C01818=1032.252,448.131,345.398,176.316,48.515,160.246
C01819=1032.229,447.887,345.444,176.296,48.510,160.242
C01820=1032.206,447.643,345.489,176.276,48.504,160.237
C01821=1032.183,447.398,345.535,176.258,48.499,160.233
C01822=1032.162,447.153,345.582,176.238,48.494,160.228
C01823=1032.140,446.909,345.629,176.219,48.489,160.224
C01824=1032.119,446.665,345.676,176.200,48.483,160.220
C01825=1032.099,446.420,345.724,176.181,48.478,160.215
C01826=1032.079,446.176,345.773,176.162,48.472,160.211
C01827=1032.060,445.932,345.821,176.143,48.467,160.206
C01828=1032.041,445.688,345.870,176.124,48.461,160.201
C01829=1032.022,445.444,345.920,176.106,48.455,160.197
C01830=1032.004,445.200,345.970,176.088,48.449,160.193
C01831=1031.987,444.957,346.020,176.069,48.443,160.188
C01832=1031.969,444.713,346.072,176.050,48.437,160.183
C01833=1031.953,444.468,346.122,176.033,48.431,160.179
C01834=1031.938,444.225,346.174,176.014,48.425,160.174
C01835=1031.921,443.982,346.226,175.996,48.419,160.170
C01836=1031.908,443.739,346.279,175.977,48.412,160.165
C01837=1031.892,443.495,346.332,175.960,48.406,160.161
C01838=1031.879,443.253,346.385,175.942,48.399,160.156
C01839=1031.864,443.010,346.438,175.924,48.393,160.152
C01840=1031.851,442.766,346.491,175.906,48.386,160.147
C01841=1031.838,442.521,346.545,175.889,48.379,160.142
C01842=1031.824,442.278,346.598,175.870,48.374,160.138
C01843=1031.810,442.034,346.652,175.853,48.367,160.133
C01844=1031.796,441.790,346.704,175.836,48.361,160.129
C01845=1031.783,441.546,346.758,175.818,48.354,160.125
C01846=1031.769,441.302,346.810,175.801,48.347,160.120
C01847=1031.755,441.058,346.864,175.784,48.341,160.116
C01848=1031.742,440.814,346.916,175.766,48.335,160.111
C01849=1031.728,440.570,346.970,175.749,48.329,160.107
C01850=1031.715,440.326,347.023,175.732,48.322,160.103
C01851=1031.702,440.082,347.075,175.715,48.316,160.098
C01852=1031.688,439.838,347.129,175.698,48.310,160.094
C01853=1031.675,439.594,347.180,175.681,48.304,160.090
C01854=1031.662,439.350,347.234,175.664,48.297,160.085
C01855=1031.648,439.106,347.286,175.646,48.291,160.081
C01856=1031.634,438.844,347.343,175.629,48.284,160.076
C01857=1031.620,438.582,347.399,175.611,48.278,160.072
C01858=1031.606,438.319,347.456,175.593,48.271,160.067
C01859=1031.591,438.057,347.511,175.575,48.265,160.063
C01860=1031.578,437.813,347.564,175.559,48.258,160.059
C01861=1031.565,437.569,347.615,175.542,48.253,160.054
C01862=1031.552,437.324,347.668,175.526,48.246,160.050
C01863=1031.539,437.080,347.720,175.509,48.241,160.046
C01864=1031.526,436.836,347.772,175.494,48.234,160.042
C01865=1031.513,436.592,347.824,175.477,48.229,160.038
C01866=1031.500,436.347,347.876,175.461,48.222,160.034
C01867=1031.487,436.103,347.928,175.444,48.217,160.030
C01868=1031.474,435.859,347.979,175.429,48.211,160.026
C01869=1031.462,435.615,348.031,175.413,48.205,160.022
C01870=1031.448,435.370,348.083,175.396,48.199,160.018
C01871=1031.436,435.126,348.134,175.381,48.193,160.014
C01872=1031.423,434.882,348.186,175.365,48.187,160.010
C01873=1031.410,434.637,348.237,175.350,48.182,160.006
C01874=1031.398,434.392,348.289,175.334,48.176,160.002
C01875=1031.385,434.149,348.340,175.317,48.170,159.998
C01876=1031.366,433.797,348.414,175.296,48.162,159.992
C01877=1031.348,433.447,348.487,175.273,48.154,159.987
C01878=1031.330,433.095,348.560,175.251,48.145,159.981
C01879=1031.312,432.744,348.634,175.229,48.137,159.976
C01880=1031.299,432.500,348.685,175.214,48.132,159.972
C01881=1031.287,432.256,348.735,175.198,48.126,159.968
C01882=1031.274,432.011,348.786,175.183,48.121,159.965
C01883=1031.262,431.766,348.837,175.168,48.115,159.961
C01884=1031.249,431.521,348.888,175.153,48.110,159.957
C01885=1031.237,431.277,348.938,175.137,48.104,159.953
C01886=1031.224,431.032,348.989,175.123,48.098,159.950
C01887=1031.212,430.788,349.039,175.108,48.093,159.946
C01888=1031.199,430.543,349.090,175.093,48.087,159.942
C01889=1031.187,430.299,349.140,175.078,48.082,159.938
C01890=1031.175,430.054,349.191,175.064,48.077,159.935
C01891=1031.163,429.809,349.242,175.049,48.071,159.931
C01892=1031.151,429.565,349.291,175.033,48.066,159.928
C01893=1031.139,429.320,349.341,175.019,48.061,159.924
C01894=1031.126,429.076,349.392,175.004,48.055,159.920
C01895=1031.114,428.831,349.442,174.990,48.050,159.917
C01896=1031.102,428.586,349.493,174.976,48.045,159.913
C01897=1031.091,428.342,349.543,174.961,48.039,159.910
C01898=1031.078,428.097,349.593,174.946,48.034,159.906
C01899=1031.066,427.852,349.643,174.933,48.029,159.903
C01900=1031.055,427.608,349.692,174.919,48.023,159.899
C01901=1031.042,427.363,349.742,174.904,48.019,159.896
C01902=1031.030,427.118,349.792,174.890,48.013,159.892
C01903=1031.019,426.874,349.842,174.876,48.008,159.889
C01904=1031.007,426.628,349.892,174.861,48.003,159.885
C01905=1030.995,426.383,349.942,174.847,47.998,159.882
C01906=1030.983,426.139,349.991,174.834,47.993,159.878
C01907=1030.971,425.893,350.040,174.819,47.988,159.875
C01908=1030.959,425.649,350.089,174.805,47.983,159.872
C01909=1030.947,425.404,350.139,174.791,47.978,159.868
C01910=1030.935,425.159,350.188,174.778,47.972,159.865
C01911=1030.923,424.914,350.238,174.764,47.967,159.861
C01912=1030.913,424.705,350.280,174.752,47.963,159.859
C01913=1030.903,424.497,350.322,174.740,47.959,159.856
C01914=1030.893,424.288,350.364,174.729,47.955,159.853
C01915=1030.883,424.079,350.406,174.717,47.950,159.850
C01916=1030.874,423.871,350.447,174.706,47.947,159.847
C01917=1030.864,423.662,350.489,174.693,47.942,159.845
C01918=1030.854,423.453,350.531,174.682,47.938,159.842
C01919=1030.844,423.244,350.572,174.671,47.934,159.839
C01920=1030.833,422.999,350.621,174.657,47.929,159.836
C01921=1030.821,422.753,350.670,174.644,47.924,159.833
C01922=1030.809,422.509,350.720,174.630,47.920,159.829
C01923=1030.797,422.264,350.767,174.617,47.914,159.826
C01924=1030.786,422.019,350.816,174.604,47.910,159.823
C01925=1030.775,421.773,350.865,174.591,47.905,159.820
C01926=1030.763,421.529,350.913,174.578,47.900,159.817
C01927=1030.751,421.283,350.962,174.564,47.896,159.813
C01928=1030.740,421.038,351.011,174.551,47.891,159.810
C01929=1030.729,420.793,351.059,174.539,47.886,159.807
C01930=1030.717,420.548,351.107,174.525,47.882,159.804
C01931=1030.705,420.303,351.156,174.512,47.877,159.801
C01932=1030.695,420.058,351.204,174.499,47.872,159.798
C01933=1030.683,419.813,351.251,174.486,47.867,159.795
C01934=1030.672,419.568,351.300,174.473,47.863,159.792
C01935=1030.661,419.323,351.348,174.461,47.858,159.789
C01936=1030.649,419.078,351.396,174.447,47.854,159.786
C01937=1030.638,418.832,351.444,174.434,47.850,159.783
C01938=1030.627,418.587,351.492,174.422,47.845,159.779
C01939=1030.616,418.342,351.539,174.409,47.841,159.777
C01940=1030.604,418.097,351.588,174.397,47.836,159.773
C01941=1030.593,417.852,351.636,174.384,47.831,159.771
C01942=1030.582,417.607,351.683,174.372,47.827,159.768
C01943=1030.571,417.361,351.731,174.359,47.822,159.765
C01944=1030.560,417.116,351.779,174.346,47.818,159.762
C01945=1030.549,416.872,351.827,174.334,47.814,159.759
C01946=1030.538,416.626,351.874,174.322,47.809,159.756
C01947=1030.527,416.380,351.923,174.310,47.805,159.753
C01948=1030.516,416.135,351.969,174.298,47.801,159.750
C01949=1030.505,415.890,352.017,174.285,47.796,159.747
C01950=1030.494,415.645,352.064,174.273,47.792,159.744
C01951=1030.483,415.399,352.111,174.261,47.788,159.741
C01952=1030.472,415.154,352.158,174.248,47.783,159.739
C01953=1030.461,414.909,352.206,174.236,47.780,159.736
C01954=1030.450,414.664,352.253,174.224,47.775,159.733
C01955=1030.439,414.418,352.300,174.212,47.771,159.730
C01956=1030.428,414.173,352.347,174.199,47.767,159.727
C01957=1030.418,413.928,352.394,174.187,47.763,159.725
C01958=1030.406,413.682,352.441,174.175,47.758,159.722
C01959=1030.396,413.437,352.488,174.164,47.754,159.719
C01960=1030.385,413.192,352.535,174.152,47.750,159.716
C01961=1030.374,412.947,352.581,174.140,47.746,159.713
C01962=1030.363,412.701,352.629,174.128,47.742,159.711
C01963=1030.352,412.456,352.676,174.116,47.737,159.708
C01964=1030.343,412.210,352.722,174.105,47.733,159.705
C01965=1030.332,411.965,352.769,174.093,47.730,159.703
C01966=1030.321,411.720,352.815,174.082,47.726,159.700
C01967=1030.310,411.473,352.862,174.070,47.722,159.697
C01968=1030.299,411.229,352.909,174.058,47.717,159.694
C01969=1030.289,410.983,352.956,174.046,47.713,159.692
C01970=1030.278,410.738,353.002,174.035,47.709,159.689
C01971=1030.268,410.492,353.049,174.023,47.705,159.686
C01972=1030.258,410.247,353.095,174.012,47.702,159.684
C01973=1030.247,410.001,353.141,174.000,47.698,159.681
C01974=1030.236,409.756,353.187,173.989,47.694,159.679
C01975=1030.226,409.510,353.233,173.977,47.690,159.676
C01976=1030.215,409.241,353.284,173.965,47.686,159.673
C01977=1030.203,408.972,353.334,173.952,47.682,159.670
C01978=1030.191,408.703,353.385,173.940,47.677,159.668
C01979=1030.180,408.433,353.435,173.928,47.674,159.665
C01980=1030.169,408.188,353.481,173.916,47.670,159.662
C01981=1030.158,407.942,353.527,173.906,47.666,159.660
C01982=1030.148,407.696,353.572,173.894,47.662,159.657
C01983=1030.137,407.451,353.618,173.883,47.659,159.655
C01984=1030.127,407.205,353.664,173.871,47.655,159.652
C01985=1030.117,406.960,353.710,173.861,47.651,159.650
C01986=1030.106,406.715,353.756,173.850,47.648,159.647
C01987=1030.096,406.468,353.802,173.838,47.644,159.645
C01988=1030.086,406.223,353.847,173.828,47.640,159.642
C01989=1030.076,405.978,353.893,173.817,47.637,159.640
C01990=1030.065,405.732,353.938,173.806,47.633,159.637
C01991=1030.055,405.487,353.984,173.795,47.629,159.635
C01992=1030.045,405.240,354.029,173.784,47.626,159.633
C01993=1030.035,404.996,354.074,173.773,47.622,159.630
C01994=1030.025,404.749,354.120,173.762,47.619,159.628
C01995=1030.015,404.504,354.165,173.752,47.615,159.625
C01996=1030.004,404.258,354.210,173.741,47.612,159.623
C01997=1029.994,404.013,354.256,173.730,47.608,159.620
C01998=1029.984,403.767,354.301,173.719,47.605,159.618
C01999=1029.974,403.522,354.346,173.709,47.601,159.616
C02000=1029.964,403.276,354.392,173.699,47.598,159.613
C02001=1029.954,403.031,354.437,173.688,47.594,159.611
C02002=1029.944,402.785,354.481,173.677,47.590,159.609
C02003=1029.934,402.539,354.527,173.666,47.588,159.606
C02004=1029.924,402.293,354.571,173.656,47.584,159.604
C02005=1029.915,402.048,354.616,173.646,47.581,159.602
C02006=1029.904,401.802,354.661,173.635,47.577,159.599
C02007=1029.894,401.556,354.706,173.625,47.574,159.597
C02008=1029.885,401.311,354.751,173.615,47.570,159.595
C02009=1029.874,401.064,354.796,173.604,47.567,159.593
C02010=1029.865,400.819,354.841,173.594,47.564,159.590
C02011=1029.855,400.573,354.886,173.583,47.560,159.588
C02012=1029.846,400.327,354.930,173.573,47.557,159.586
C02013=1029.835,400.082,354.974,173.563,47.554,159.584
C02014=1029.825,399.836,355.019,173.552,47.550,159.581
C02015=1029.815,399.590,355.064,173.542,47.547,159.579
C02016=1029.806,399.344,355.108,173.531,47.544,159.577
C02017=1029.795,399.099,355.153,173.521,47.541,159.575
C02018=1029.786,398.853,355.197,173.512,47.538,159.572
C02019=1029.776,398.607,355.242,173.502,47.535,159.570
C02020=1029.767,398.361,355.286,173.492,47.532,159.568
C02021=1029.757,398.115,355.329,173.482,47.528,159.566
C02022=1029.747,397.870,355.374,173.471,47.525,159.564
C02023=1029.737,397.624,355.418,173.461,47.523,159.562
C02024=1029.727,397.378,355.462,173.451,47.520,159.560
C02025=1029.718,397.132,355.506,173.441,47.516,159.557
C02026=1029.707,396.886,355.550,173.431,47.513,159.555
C02027=1029.698,396.640,355.594,173.422,47.510,159.553
C02028=1029.689,396.394,355.638,173.412,47.507,159.551
C02029=1029.678,396.148,355.682,173.402,47.504,159.549
C02030=1029.670,395.903,355.725,173.392,47.501,159.547
C02031=1029.660,395.657,355.770,173.382,47.498,159.545
C02032=1029.650,395.411,355.813,173.373,47.495,159.543
C02033=1029.641,395.165,355.857,173.363,47.492,159.541
C02034=1029.631,394.919,355.901,173.353,47.490,159.539
C02035=1029.622,394.674,355.944,173.343,47.486,159.536
C02036=1029.611,394.425,355.989,173.334,47.484,159.534
C02037=1029.602,394.178,356.033,173.324,47.480,159.532
C02038=1029.593,393.930,356.077,173.314,47.478,159.530
C02039=1029.583,393.683,356.120,173.304,47.475,159.528
C02040=1029.574,393.436,356.164,173.295,47.472,159.526
C02041=1029.564,393.190,356.207,173.285,47.469,159.524
C02042=1029.555,392.944,356.250,173.276,47.467,159.522
C02043=1029.545,392.698,356.294,173.266,47.464,159.520
C02044=1029.535,392.452,356.337,173.256,47.461,159.518
C02045=1029.527,392.206,356.380,173.247,47.459,159.516
C02046=1029.517,391.960,356.423,173.238,47.455,159.514
C02047=1029.508,391.714,356.467,173.228,47.452,159.512
C02048=1029.498,391.468,356.510,173.219,47.450,159.510
C02049=1029.489,391.223,356.554,173.209,47.447,159.508
C02050=1029.479,390.976,356.596,173.200,47.445,159.506
C02051=1029.470,390.730,356.639,173.191,47.442,159.505
C02052=1029.461,390.484,356.683,173.182,47.439,159.503
C02053=1029.452,390.239,356.725,173.172,47.436,159.501
C02054=1029.442,389.992,356.769,173.162,47.434,159.499
C02055=1029.433,389.746,356.811,173.154,47.431,159.497
C02056=1029.423,389.500,356.854,173.145,47.429,159.495
C02057=1029.415,389.254,356.897,173.135,47.426,159.493
C02058=1029.405,389.007,356.940,173.126,47.423,159.491
C02059=1029.396,388.761,356.982,173.117,47.421,159.489
C02060=1029.387,388.516,357.025,173.108,47.418,159.487
C02061=1029.377,388.269,357.068,173.098,47.416,159.486
C02062=1029.368,388.023,357.110,173.090,47.413,159.484
C02063=1029.359,387.777,357.153,173.080,47.411,159.482
C02064=1029.350,387.531,357.196,173.072,47.408,159.480
C02065=1029.341,387.285,357.239,173.063,47.406,159.478
C02066=1029.332,387.038,357.280,173.053,47.403,159.476
C02067=1029.322,386.793,357.323,173.045,47.401,159.475
C02068=1029.313,386.546,357.366,173.036,47.399,159.473
C02069=1029.304,386.300,357.408,173.027,47.396,159.471
C02070=1029.295,386.054,357.450,173.018,47.393,159.469
C02071=1029.286,385.807,357.492,173.008,47.391,159.467
C02072=1029.276,385.561,357.535,173.000,47.389,159.466
C02073=1029.267,385.315,357.577,172.991,47.387,159.464
C02074=1029.258,385.069,357.619,172.983,47.384,159.462
C02075=1029.249,384.823,357.661,172.973,47.382,159.460
C02076=1029.240,384.576,357.702,172.965,47.380,159.459
C02077=1029.231,384.330,357.745,172.956,47.377,159.457
C02078=1029.222,384.084,357.787,172.948,47.375,159.455
C02079=1029.213,383.838,357.828,172.938,47.373,159.453
C02080=1029.203,383.591,357.871,172.930,47.371,159.452
C02081=1029.194,383.345,357.913,172.921,47.368,159.450
C02082=1029.186,383.099,357.955,172.913,47.366,159.448
C02083=1029.177,382.852,357.996,172.903,47.364,159.446
C02084=1029.168,382.606,358.038,172.895,47.361,159.445
C02085=1029.159,382.359,358.080,172.887,47.359,159.443
C02086=1029.150,382.113,358.121,172.878,47.357,159.442
C02087=1029.141,381.867,358.163,172.870,47.355,159.440
C02088=1029.133,381.621,358.205,172.860,47.353,159.438
C02089=1029.124,381.375,358.246,172.852,47.350,159.436
C02090=1029.115,381.128,358.288,172.844,47.348,159.435
C02091=1029.106,380.882,358.330,172.835,47.346,159.433
C02092=1029.097,380.653,358.369,172.827,47.344,159.432
C02093=1029.089,380.424,358.407,172.819,47.343,159.430
C02094=1029.081,380.196,358.446,172.812,47.340,159.429
C02095=1029.072,379.967,358.484,172.804,47.339,159.427
C02096=1029.065,379.737,358.522,172.796,47.337,159.426
C02097=1029.056,379.509,358.561,172.788,47.335,159.424
C02098=1029.048,379.279,358.599,172.780,47.332,159.422
C02099=1029.040,379.050,358.638,172.772,47.331,159.421
C02100=1029.031,378.804,358.679,172.764,47.329,159.419
C02101=1029.022,378.557,358.721,172.756,47.327,159.418
C02102=1029.014,378.311,358.762,172.748,47.324,159.416
C02103=1029.005,378.065,358.803,172.739,47.323,159.415
C02104=1028.996,377.818,358.845,172.731,47.321,159.413
C02105=1028.988,377.572,358.886,172.723,47.318,159.411
C02106=1028.979,377.326,358.927,172.715,47.317,159.410
C02107=1028.971,377.079,358.968,172.707,47.315,159.408
C02108=1028.962,376.832,359.009,172.698,47.313,159.407
C02109=1028.953,376.586,359.050,172.690,47.311,159.405
C02110=1028.944,376.339,359.091,172.682,47.309,159.404
C02111=1028.936,376.094,359.131,172.674,47.307,159.402
C02112=1028.927,375.847,359.172,172.666,47.306,159.401
C02113=1028.918,375.600,359.213,172.658,47.304,159.399
C02114=1028.909,375.354,359.254,172.650,47.302,159.398
C02115=1028.901,375.107,359.295,172.642,47.300,159.396
C02116=1028.893,374.861,359.336,172.634,47.298,159.395
C02117=1028.883,374.614,359.376,172.626,47.296,159.393
C02118=1028.875,374.368,359.417,172.618,47.294,159.392
C02119=1028.867,374.121,359.458,172.610,47.293,159.390
C02120=1028.858,373.875,359.498,172.602,47.291,159.389
C02121=1028.849,373.628,359.539,172.594,47.289,159.387
C02122=1028.840,373.382,359.579,172.586,47.288,159.386
C02123=1028.832,373.135,359.620,172.578,47.286,159.384
C02124=1028.824,372.889,359.660,172.570,47.284,159.383
C02125=1028.815,372.641,359.700,172.562,47.282,159.381
C02126=1028.807,372.395,359.741,172.554,47.281,159.380
C02127=1028.799,372.149,359.781,172.546,47.279,159.378
C02128=1028.789,371.902,359.822,172.538,47.277,159.377
C02129=1028.781,371.656,359.862,172.531,47.276,159.376
C02130=1028.774,371.409,359.902,172.523,47.274,159.374
C02131=1028.764,371.162,359.943,172.515,47.273,159.373
C02132=1028.756,370.916,359.983,172.507,47.271,159.371
C02133=1028.748,370.669,360.023,172.500,47.269,159.370
C02134=1028.740,370.423,360.063,172.492,47.267,159.368
C02135=1028.731,370.176,360.104,172.484,47.266,159.367
C02136=1028.723,369.930,360.144,172.476,47.264,159.366
C02137=1028.715,369.683,360.184,172.469,47.263,159.364
C02138=1028.706,369.437,360.224,172.462,47.261,159.363
C02139=1028.698,369.190,360.264,172.454,47.259,159.361
C02140=1028.690,368.943,360.304,172.447,47.258,159.360
C02141=1028.681,368.696,360.344,172.439,47.256,159.359
C02142=1028.673,368.450,360.384,172.431,47.255,159.357
C02143=1028.665,368.203,360.424,172.423,47.253,159.356
C02144=1028.656,367.956,360.463,172.416,47.252,159.355
C02145=1028.647,367.709,360.503,172.408,47.251,159.353
C02146=1028.639,367.463,360.542,172.400,47.249,159.352
C02147=1028.631,367.217,360.583,172.393,47.248,159.351
C02148=1028.622,366.970,360.622,172.385,47.246,159.349
C02149=1028.614,366.723,360.661,172.378,47.245,159.348
C02150=1028.606,366.477,360.701,172.371,47.243,159.347
C02151=1028.598,366.230,360.741,172.363,47.242,159.345
C02152=1028.590,366.011,360.775,172.357,47.241,159.344
C02153=1028.583,365.792,360.811,172.350,47.239,159.343
C02154=1028.575,365.574,360.845,172.343,47.239,159.342
C02155=1028.568,365.356,360.880,172.337,47.238,159.341
C02156=1028.561,365.137,360.916,172.330,47.236,159.340
C02157=1028.553,364.919,360.951,172.324,47.235,159.339
C02158=1028.546,364.701,360.985,172.317,47.233,159.337
C02159=1028.539,364.482,361.020,172.311,47.232,159.336
C02160=1028.531,364.235,361.060,172.303,47.231,159.335
C02161=1028.522,363.988,361.099,172.296,47.230,159.334
C02162=1028.515,363.742,361.139,172.289,47.229,159.333
C02163=1028.506,363.494,361.177,172.282,47.227,159.331
C02164=1028.498,363.248,361.217,172.274,47.226,159.330
C02165=1028.490,363.002,361.256,172.267,47.225,159.329
C02166=1028.483,362.754,361.295,172.260,47.224,159.328
C02167=1028.474,362.508,361.334,172.253,47.222,159.326
C02168=1028.466,362.261,361.373,172.245,47.221,159.325
C02169=1028.458,362.014,361.413,172.238,47.220,159.324
C02170=1028.450,361.767,361.452,172.231,47.219,159.323
C02171=1028.442,361.521,361.491,172.224,47.217,159.321
C02172=1028.434,361.274,361.530,172.217,47.217,159.320
C02173=1028.426,361.027,361.570,172.210,47.215,159.319
C02174=1028.418,360.780,361.608,172.203,47.214,159.318
C02175=1028.410,360.533,361.647,172.195,47.213,159.316
C02176=1028.402,360.287,361.686,172.189,47.212,159.315
C02177=1028.394,360.039,361.724,172.181,47.211,159.314
C02178=1028.385,359.793,361.764,172.174,47.210,159.313
C02179=1028.377,359.546,361.802,172.167,47.208,159.312
C02180=1028.370,359.299,361.840,172.160,47.207,159.311
C02181=1028.362,359.052,361.879,172.153,47.207,159.309
C02182=1028.353,358.805,361.918,172.146,47.205,159.308
C02183=1028.346,358.559,361.957,172.139,47.204,159.307
C02184=1028.337,358.312,361.995,172.132,47.204,159.306
C02185=1028.329,358.064,362.034,172.125,47.202,159.305
C02186=1028.322,357.818,362.072,172.118,47.201,159.304
C02187=1028.314,357.571,362.111,172.111,47.200,159.303
C02188=1028.305,357.323,362.149,172.104,47.199,159.301
C02189=1028.298,357.077,362.188,172.097,47.199,159.300
C02190=1028.290,356.830,362.226,172.091,47.198,159.299
C02191=1028.282,356.583,362.264,172.083,47.196,159.298
C02192=1028.273,356.336,362.302,172.077,47.195,159.297
C02193=1028.265,356.089,362.341,172.069,47.195,159.296
C02194=1028.258,355.843,362.379,172.063,47.193,159.295
C02195=1028.249,355.595,362.418,172.056,47.193,159.294
C02196=1028.242,355.349,362.456,172.050,47.192,159.293
C02197=1028.234,355.102,362.495,172.042,47.191,159.291
C02198=1028.226,354.854,362.532,172.036,47.190,159.290
C02199=1028.218,354.607,362.571,172.029,47.189,159.289
C02200=1028.210,354.361,362.609,172.021,47.188,159.288
C02201=1028.202,354.114,362.647,172.015,47.187,159.287
C02202=1028.195,353.867,362.685,172.008,47.187,159.286
C02203=1028.186,353.619,362.723,172.002,47.186,159.285
C02204=1028.178,353.373,362.760,171.995,47.185,159.284
C02205=1028.171,353.126,362.798,171.988,47.184,159.283
C02206=1028.163,352.879,362.837,171.981,47.184,159.282
C02207=1028.156,352.632,362.875,171.975,47.183,159.281
C02208=1028.147,352.385,362.913,171.968,47.182,159.280
C02209=1028.139,352.138,362.950,171.962,47.181,159.279
C02210=1028.132,351.891,362.988,171.955,47.180,159.278
C02211=1028.124,351.643,363.026,171.948,47.180,159.277
C02212=1028.117,351.429,363.059,171.942,47.179,159.276
C02213=1028.111,351.213,363.092,171.937,47.178,159.275
C02214=1028.103,350.998,363.125,171.931,47.178,159.274
C02215=1028.097,350.782,363.158,171.925,47.178,159.273
C02216=1028.090,350.568,363.190,171.919,47.177,159.272
C02217=1028.083,350.352,363.223,171.914,47.176,159.271
C02218=1028.076,350.137,363.256,171.908,47.175,159.270
C02219=1028.070,349.922,363.289,171.902,47.175,159.269
C02220=1028.063,349.675,363.327,171.896,47.174,159.269
C02221=1028.054,349.428,363.364,171.890,47.173,159.268
C02222=1028.047,349.180,363.402,171.882,47.173,159.266
C02223=1028.040,348.933,363.439,171.877,47.172,159.266
C02224=1028.032,348.686,363.476,171.870,47.172,159.265
C02225=1028.024,348.440,363.515,171.863,47.171,159.264
C02226=1028.015,348.192,363.552,171.857,47.171,159.263
C02227=1028.008,347.945,363.589,171.850,47.170,159.262
C02228=1028.000,347.698,363.626,171.844,47.169,159.261
C02229=1027.993,347.451,363.664,171.838,47.169,159.260
C02230=1027.985,347.204,363.701,171.831,47.168,159.259
C02231=1027.977,346.957,363.739,171.825,47.168,159.258
C02232=1027.969,346.710,363.776,171.819,47.167,159.257
C02233=1027.962,346.463,363.813,171.812,47.166,159.256
C02234=1027.954,346.215,363.849,171.806,47.166,159.255
C02235=1027.947,345.968,363.887,171.800,47.166,159.254
C02236=1027.939,345.721,363.924,171.793,47.165,159.253
C02237=1027.932,345.474,363.961,171.787,47.165,159.252
C02238=1027.924,345.227,363.998,171.780,47.164,159.251
C02239=1027.917,344.980,364.036,171.774,47.164,159.250
C02240=1027.909,344.733,364.072,171.768,47.163,159.249
C02241=1027.901,344.486,364.109,171.762,47.163,159.249
C02242=1027.894,344.239,364.146,171.755,47.163,159.248
C02243=1027.886,343.991,364.183,171.749,47.162,159.247
C02244=1027.879,343.744,364.220,171.743,47.162,159.246
C02245=1027.871,343.497,364.257,171.737,47.161,159.245
C02246=1027.864,343.250,364.294,171.730,47.161,159.244
C02247=1027.856,343.003,364.331,171.724,47.161,159.243
C02248=1027.848,342.755,364.367,171.718,47.160,159.242
C02249=1027.841,342.508,364.405,171.712,47.160,159.241
C02250=1027.833,342.261,364.442,171.705,47.160,159.241
C02251=1027.825,342.014,364.478,171.699,47.159,159.240
C02252=1027.818,341.766,364.515,171.693,47.159,159.239
C02253=1027.810,341.519,364.552,171.687,47.158,159.238
C02254=1027.803,341.272,364.588,171.681,47.158,159.237
C02255=1027.795,341.025,364.625,171.674,47.158,159.236
C02256=1027.788,340.777,364.661,171.668,47.157,159.235
C02257=1027.780,340.531,364.698,171.662,47.157,159.234
C02258=1027.773,340.283,364.735,171.656,47.157,159.234
C02259=1027.766,340.036,364.771,171.651,47.156,159.233
C02260=1027.758,339.789,364.807,171.644,47.156,159.232
C02261=1027.750,339.542,364.844,171.638,47.156,159.231
C02262=1027.742,339.294,364.880,171.632,47.156,159.230
C02263=1027.735,339.048,364.916,171.626,47.155,159.229
C02264=1027.728,338.800,364.953,171.620,47.155,159.229
C02265=1027.721,338.552,364.989,171.613,47.155,159.228
C02266=1027.713,338.305,365.026,171.607,47.155,159.227
C02267=1027.705,338.057,365.062,171.602,47.155,159.226
C02268=1027.698,337.811,365.098,171.596,47.155,159.225
C02269=1027.690,337.564,365.135,171.590,47.154,159.225
C02270=1027.683,337.316,365.171,171.584,47.154,159.224
C02271=1027.675,337.069,365.207,171.577,47.154,159.223
C02272=1027.669,336.852,365.238,171.573,47.154,159.222
C02273=1027.662,336.636,365.270,171.567,47.154,159.222
C02274=1027.656,336.418,365.302,171.562,47.154,159.221
C02275=1027.649,336.202,365.333,171.556,47.154,159.220
C02276=1027.643,335.985,365.366,171.552,47.153,159.219
C02277=1027.637,335.768,365.396,171.546,47.154,159.219
C02278=1027.630,335.552,365.429,171.541,47.154,159.218
C02279=1027.624,335.334,365.460,171.536,47.154,159.217
C02280=1027.616,335.087,365.496,171.530,47.153,159.217
C02281=1027.610,334.840,365.532,171.524,47.153,159.216
C02282=1027.602,334.592,365.568,171.518,47.154,159.215
C02283=1027.595,334.346,365.604,171.512,47.153,159.214
C02284=1027.587,334.098,365.640,171.507,47.153,159.214
C02285=1027.580,333.850,365.676,171.501,47.153,159.213
C02286=1027.573,333.603,365.712,171.495,47.153,159.212
C02287=1027.565,333.355,365.747,171.490,47.153,159.211
C02288=1027.558,333.109,365.783,171.484,47.153,159.211
C02289=1027.550,332.861,365.819,171.478,47.153,159.210
C02290=1027.543,332.614,365.854,171.472,47.153,159.209
C02291=1027.535,332.367,365.890,171.466,47.153,159.208
C02292=1027.529,332.119,365.925,171.460,47.153,159.208
C02293=1027.521,331.872,365.962,171.454,47.154,159.207
C02294=1027.514,331.624,365.997,171.449,47.154,159.206
C02295=1027.506,331.377,366.032,171.443,47.153,159.205
C02296=1027.499,331.130,366.067,171.437,47.153,159.205
C02297=1027.491,330.883,366.104,171.431,47.154,159.204
C02298=1027.485,330.635,366.139,171.426,47.154,159.203
C02299=1027.477,330.388,366.175,171.420,47.154,159.203
C02300=1027.470,330.140,366.210,171.414,47.154,159.202
C02301=1027.462,329.893,366.245,171.409,47.154,159.201
C02302=1027.455,329.646,366.281,171.403,47.154,159.201
C02303=1027.448,329.398,366.316,171.397,47.154,159.200
C02304=1027.441,329.150,366.352,171.392,47.155,159.199
C02305=1027.434,328.904,366.387,171.386,47.155,159.199
C02306=1027.426,328.656,366.422,171.380,47.155,159.198
C02307=1027.419,328.409,366.457,171.375,47.155,159.197
C02308=1027.412,328.161,366.493,171.369,47.155,159.197
C02309=1027.404,327.914,366.529,171.363,47.155,159.196
C02310=1027.398,327.666,366.564,171.358,47.155,159.195
C02311=1027.390,327.419,366.598,171.352,47.156,159.194
C02312=1027.383,327.171,366.634,171.347,47.156,159.194
C02313=1027.375,326.924,366.668,171.341,47.157,159.193
C02314=1027.368,326.677,366.704,171.336,47.157,159.193
C02315=1027.360,326.429,366.739,171.330,47.157,159.192
C02316=1027.353,326.182,366.773,171.325,47.158,159.191
C02317=1027.346,325.935,366.808,171.319,47.158,159.191
C02318=1027.338,325.687,366.843,171.313,47.158,159.190
C02319=1027.331,325.440,366.878,171.308,47.159,159.190
C02320=1027.324,325.192,366.912,171.302,47.159,159.189
C02321=1027.316,324.944,366.947,171.297,47.159,159.188
C02322=1027.309,324.697,366.982,171.291,47.160,159.188
C02323=1027.302,324.450,367.017,171.286,47.160,159.187
C02324=1027.295,324.202,367.052,171.280,47.161,159.186
C02325=1027.287,323.954,367.086,171.275,47.161,159.186
C02326=1027.280,323.707,367.120,171.269,47.161,159.185
C02327=1027.273,323.460,367.156,171.264,47.162,159.185
C02328=1027.265,323.213,367.190,171.258,47.162,159.184
C02329=1027.259,322.965,367.225,171.253,47.163,159.183
C02330=1027.251,322.717,367.259,171.247,47.163,159.183
C02331=1027.243,322.470,367.294,171.243,47.163,159.182
C02332=1027.237,322.250,367.325,171.237,47.163,159.182
C02333=1027.231,322.031,367.356,171.233,47.164,159.181
C02334=1027.224,321.812,367.386,171.227,47.165,159.181
C02335=1027.218,321.593,367.416,171.223,47.165,159.180
C02336=1027.211,321.374,367.447,171.218,47.165,159.180
C02337=1027.205,321.155,367.478,171.213,47.166,159.179
C02338=1027.200,320.936,367.508,171.209,47.166,159.179
C02339=1027.192,320.718,367.538,171.204,47.167,159.178
C02340=1027.186,320.470,367.573,171.199,47.167,159.177
C02341=1027.179,320.223,367.607,171.193,47.168,159.177
C02342=1027.171,319.975,367.641,171.188,47.168,159.176
C02343=1027.164,319.727,367.677,171.182,47.168,159.176
C02344=1027.157,319.479,367.710,171.177,47.169,159.175
C02345=1027.150,319.232,367.746,171.171,47.169,159.175
C02346=1027.143,318.984,367.779,171.167,47.170,159.174
C02347=1027.136,318.736,367.813,171.162,47.171,159.174
C02348=1027.129,318.489,367.848,171.156,47.171,159.173
C02349=1027.122,318.241,367.882,171.150,47.171,159.172
C02350=1027.114,317.994,367.917,171.145,47.172,159.172
C02351=1027.108,317.747,367.951,171.140,47.173,159.171
C02352=1027.101,317.499,367.985,171.135,47.173,159.171
C02353=1027.094,317.252,368.019,171.130,47.174,159.170
C02354=1027.087,317.004,368.054,171.124,47.174,159.170
C02355=1027.080,316.757,368.087,171.119,47.175,159.169
C02356=1027.073,316.509,368.121,171.113,47.175,159.169
C02357=1027.066,316.262,368.156,171.108,47.176,159.168
C02358=1027.059,316.014,368.190,171.104,47.176,159.168
C02359=1027.052,315.766,368.224,171.098,47.177,159.167
C02360=1027.046,315.519,368.258,171.093,47.178,159.167
C02361=1027.038,315.272,368.293,171.088,47.179,159.166
C02362=1027.031,315.024,368.326,171.082,47.180,159.166
C02363=1027.024,314.776,368.361,171.078,47.179,159.165
C02364=1027.017,314.529,368.395,171.072,47.180,159.164
C02365=1027.010,314.281,368.428,171.067,47.181,159.164
C02366=1027.004,314.034,368.463,171.062,47.182,159.163
C02367=1026.997,313.786,368.496,171.057,47.182,159.163
C02368=1026.990,313.538,368.530,171.052,47.183,159.162
C02369=1026.983,313.291,368.565,171.047,47.184,159.162
C02370=1026.976,313.044,368.599,171.041,47.184,159.161
C02371=1026.969,312.796,368.633,171.037,47.185,159.161
C02372=1026.963,312.548,368.667,171.032,47.186,159.160
C02373=1026.956,312.301,368.701,171.026,47.186,159.160
C02374=1026.949,312.054,368.734,171.021,47.187,159.159
C02375=1026.943,311.806,368.769,171.017,47.188,159.159
C02376=1026.935,311.558,368.803,171.011,47.188,159.158
C02377=1026.929,311.311,368.836,171.006,47.189,159.158
C02378=1026.922,311.063,368.869,171.000,47.190,159.157
C02379=1026.916,310.816,368.903,170.996,47.190,159.157
C02380=1026.909,310.568,368.937,170.991,47.191,159.157
C02381=1026.901,310.321,368.970,170.986,47.193,159.156
C02382=1026.894,310.072,369.003,170.980,47.193,159.156
C02383=1026.887,309.825,369.037,170.976,47.194,159.155
C02384=1026.879,309.578,369.070,170.971,47.195,159.155
C02385=1026.873,309.330,369.103,170.966,47.196,159.154
C02386=1026.866,309.083,369.137,170.960,47.197,159.154
C02387=1026.858,308.835,369.169,170.955,47.198,159.154
C02388=1026.851,308.587,369.203,170.951,47.199,159.153
C02389=1026.845,308.339,369.236,170.946,47.200,159.153
C02390=1026.837,308.092,369.269,170.941,47.201,159.152
C02391=1026.830,307.844,369.302,170.935,47.201,159.152
C02392=1026.824,307.628,369.331,170.931,47.203,159.152
C02393=1026.817,307.411,369.360,170.927,47.203,159.151
C02394=1026.812,307.194,369.389,170.923,47.204,159.151
C02395=1026.805,306.977,369.418,170.918,47.205,159.150
C02396=1026.799,306.761,369.447,170.914,47.206,159.150
C02397=1026.794,306.545,369.476,170.909,47.207,159.150
C02398=1026.787,306.328,369.505,170.905,47.208,159.149
C02399=1026.781,306.112,369.534,170.901,47.209,159.149
C02400=1026.774,305.864,369.566,170.896,47.209,159.149
C02401=1026.767,305.617,369.600,170.892,47.211,159.148
C02402=1026.760,305.368,369.633,170.886,47.211,159.148
C02403=1026.753,305.121,369.665,170.881,47.213,159.147
C02404=1026.746,304.873,369.699,170.877,47.213,159.147
C02405=1026.740,304.626,369.732,170.872,47.215,159.147
C02406=1026.732,304.378,369.764,170.867,47.215,159.146
C02407=1026.726,304.130,369.797,170.861,47.217,159.146
C02408=1026.719,303.883,369.831,170.857,47.218,159.146
C02409=1026.712,303.635,369.863,170.852,47.219,159.145
C02410=1026.705,303.387,369.896,170.847,47.220,159.145
C02411=1026.698,303.139,369.929,170.843,47.220,159.144
C02412=1026.691,302.891,369.961,170.838,47.222,159.144
C02413=1026.684,302.644,369.995,170.833,47.223,159.144
C02414=1026.677,302.396,370.028,170.828,47.224,159.143
C02415=1026.670,302.149,370.060,170.823,47.225,159.143
C02416=1026.664,301.901,370.093,170.818,47.226,159.142
C02417=1026.657,301.653,370.126,170.814,47.227,159.142
C02418=1026.650,301.406,370.158,170.809,47.228,159.142
C02419=1026.643,301.157,370.191,170.804,47.230,159.141
C02420=1026.637,300.910,370.224,170.800,47.231,159.141
C02421=1026.630,300.662,370.256,170.794,47.232,159.141
C02422=1026.623,300.414,370.289,170.789,47.233,159.140
C02423=1026.617,300.167,370.322,170.785,47.234,159.140
C02424=1026.610,299.919,370.354,170.780,47.235,159.140
C02425=1026.603,299.671,370.387,170.776,47.236,159.139
C02426=1026.596,299.423,370.420,170.771,47.237,159.139
C02427=1026.589,299.176,370.452,170.766,47.239,159.139
C02428=1026.582,298.928,370.485,170.762,47.240,159.138
C02429=1026.576,298.680,370.518,170.757,47.241,159.138
C02430=1026.569,298.433,370.550,170.751,47.242,159.137
C02431=1026.562,298.185,370.583,170.747,47.243,159.137
C02432=1026.556,297.937,370.616,170.742,47.244,159.137
C02433=1026.549,297.690,370.648,170.738,47.246,159.137
C02434=1026.543,297.442,370.680,170.733,47.247,159.136
C02435=1026.536,297.193,370.713,170.728,47.248,159.136
C02436=1026.529,296.946,370.745,170.724,47.249,159.136
C02437=1026.523,296.698,370.778,170.719,47.250,159.135
C02438=1026.516,296.451,370.810,170.715,47.251,159.135
C02439=1026.510,296.203,370.842,170.710,47.253,159.135
C02440=1026.503,295.955,370.875,170.706,47.254,159.134
C02441=1026.496,295.707,370.908,170.701,47.255,159.134
C02442=1026.489,295.460,370.940,170.696,47.257,159.134
C02443=1026.483,295.212,370.972,170.692,47.258,159.133
C02444=1026.476,294.964,371.004,170.687,47.259,159.133
C02445=1026.470,294.717,371.037,170.682,47.260,159.133
C02446=1026.464,294.468,371.070,170.677,47.262,159.132
C02447=1026.457,294.220,371.102,170.673,47.263,159.132
C02448=1026.450,293.973,371.134,170.668,47.264,159.132
C02449=1026.444,293.725,371.166,170.664,47.265,159.131
C02450=1026.437,293.478,371.198,170.659,47.267,159.131
C02451=1026.431,293.229,371.230,170.654,47.268,159.131
C02452=1026.419,292.813,371.284,170.647,47.270,159.131
C02453=1026.407,292.398,371.337,170.639,47.273,159.130
C02454=1026.396,291.982,371.391,170.631,47.275,159.129
C02455=1026.385,291.566,371.445,170.625,47.278,159.129
C02456=1026.378,291.318,371.476,170.620,47.279,159.129
C02457=1026.371,291.070,371.508,170.614,47.280,159.128
C02458=1026.365,290.823,371.540,170.611,47.282,159.128
C02459=1026.358,290.574,371.572,170.606,47.283,159.128
C02460=1026.351,290.326,371.604,170.602,47.285,159.128
C02461=1026.344,290.078,371.635,170.597,47.287,159.128
C02462=1026.337,289.831,371.667,170.593,47.288,159.127
C02463=1026.330,289.583,371.699,170.588,47.289,159.127
C02464=1026.324,289.335,371.731,170.584,47.291,159.127
C02465=1026.318,289.087,371.762,170.579,47.292,159.127
C02466=1026.311,288.839,371.794,170.574,47.294,159.126
C02467=1026.304,288.591,371.825,170.570,47.295,159.126
C02468=1026.297,288.344,371.857,170.565,47.297,159.126
C02469=1026.291,288.096,371.889,170.561,47.298,159.126
C02470=1026.284,287.848,371.920,170.556,47.300,159.125
C02471=1026.277,287.600,371.951,170.552,47.301,159.125
C02472=1026.271,287.352,371.983,170.548,47.303,159.125
C02473=1026.264,287.104,372.015,170.544,47.304,159.125
C02474=1026.258,286.856,372.046,170.539,47.306,159.125
C02475=1026.251,286.608,372.078,170.535,47.307,159.124
C02476=1026.244,286.360,372.109,170.530,47.309,159.124
C02477=1026.237,286.113,372.141,170.526,47.310,159.124
C02478=1026.231,285.865,372.172,170.521,47.312,159.124
C02479=1026.224,285.617,372.203,170.516,47.314,159.123
C02480=1026.217,285.369,372.235,170.513,47.316,159.123
C02481=1026.211,285.121,372.266,170.508,47.317,159.123
C02482=1026.204,284.873,372.298,170.504,47.319,159.123
C02483=1026.197,284.625,372.329,170.499,47.321,159.123
C02484=1026.190,284.377,372.359,170.495,47.322,159.122
C02485=1026.184,284.130,372.390,170.490,47.324,159.122
C02486=1026.177,283.882,372.422,170.487,47.326,159.122
C02487=1026.170,283.634,372.453,170.482,47.327,159.122
C02488=1026.164,283.385,372.484,170.478,47.329,159.122
C02489=1026.157,283.138,372.515,170.473,47.331,159.122
C02490=1026.151,282.890,372.547,170.469,47.332,159.121
C02491=1026.143,282.642,372.578,170.464,47.334,159.121
C02492=1026.137,282.393,372.608,170.461,47.336,159.121
C02493=1026.130,282.146,372.640,170.456,47.337,159.121
C02494=1026.123,281.898,372.671,170.452,47.339,159.121
C02495=1026.117,281.650,372.702,170.447,47.341,159.120
C02496=1026.111,281.402,372.733,170.443,47.343,159.120
C02497=1026.104,281.154,372.764,170.438,47.344,159.120
C02498=1026.097,280.906,372.795,170.435,47.346,159.120
C02499=1026.090,280.658,372.826,170.430,47.348,159.120
C02500=1026.083,280.410,372.857,170.426,47.349,159.120
C02501=1026.077,280.162,372.888,170.421,47.352,159.120
C02502=1026.071,279.914,372.919,170.417,47.353,159.119
C02503=1026.064,279.666,372.950,170.413,47.355,159.119
C02504=1026.058,279.418,372.981,170.409,47.356,159.119
C02505=1026.051,279.170,373.011,170.404,47.358,159.119
C02506=1026.044,278.922,373.043,170.400,47.360,159.119
C02507=1026.038,278.674,373.073,170.395,47.362,159.118
C02508=1026.028,278.270,373.124,170.389,47.365,159.118
C02509=1026.017,277.867,373.174,170.382,47.367,159.118
C02510=1026.007,277.463,373.224,170.375,47.371,159.118
C02511=1025.996,277.060,373.274,170.368,47.373,159.118
C02512=1025.988,276.812,373.305,170.364,47.375,159.117
C02513=1025.982,276.564,373.336,170.360,47.377,159.117
C02514=1025.975,276.315,373.367,170.356,47.379,159.117
C02515=1025.969,276.068,373.396,170.351,47.381,159.117
C02516=1025.962,275.819,373.427,170.347,47.383,159.117
C02517=1025.955,275.571,373.458,170.343,47.385,159.117
C02518=1025.949,275.324,373.488,170.339,47.387,159.117
C02519=1025.943,275.075,373.519,170.334,47.389,159.117
C02520=1025.935,274.827,373.549,170.331,47.391,159.117
C02521=1025.929,274.579,373.581,170.326,47.393,159.116
C02522=1025.922,274.332,373.610,170.322,47.395,159.116
C02523=1025.916,274.083,373.641,170.319,47.397,159.116
C02524=1025.910,273.835,373.671,170.314,47.399,159.116
C02525=1025.903,273.587,373.702,170.310,47.400,159.116
C02526=1025.896,273.338,373.732,170.305,47.402,159.116
C02527=1025.890,273.092,373.763,170.302,47.404,159.116
C02528=1025.883,272.843,373.793,170.297,47.406,159.116
C02529=1025.876,272.595,373.824,170.293,47.409,159.116
C02530=1025.870,272.347,373.854,170.289,47.411,159.115
C02531=1025.863,272.099,373.884,170.285,47.412,159.115
C02532=1025.857,271.851,373.914,170.281,47.414,159.115
C02533=1025.850,271.603,373.945,170.277,47.416,159.115
C02534=1025.844,271.354,373.975,170.273,47.419,159.115
C02535=1025.837,271.107,374.005,170.268,47.421,159.115
C02536=1025.831,270.858,374.036,170.265,47.422,159.115
C02537=1025.824,270.611,374.065,170.260,47.424,159.115
C02538=1025.818,270.362,374.096,170.256,47.427,159.115
C02539=1025.811,270.115,374.126,170.252,47.429,159.115
C02540=1025.805,269.866,374.157,170.248,47.431,159.115
C02541=1025.797,269.618,374.187,170.244,47.432,159.114
C02542=1025.791,269.370,374.216,170.240,47.435,159.114
C02543=1025.785,269.121,374.247,170.236,47.437,159.114
C02544=1025.778,268.874,374.276,170.231,47.439,159.114
C02545=1025.771,268.626,374.306,170.228,47.441,159.114
C02546=1025.765,268.378,374.337,170.223,47.443,159.114
C02547=1025.758,268.129,374.367,170.220,47.446,159.114
C02548=1025.752,267.881,374.396,170.216,47.447,159.114
C02549=1025.745,267.633,374.427,170.211,47.450,159.114
C02550=1025.739,267.385,374.456,170.208,47.452,159.114
C02551=1025.732,267.137,374.487,170.203,47.454,159.114
C02552=1025.726,266.889,374.516,170.200,47.456,159.114
C02553=1025.719,266.640,374.546,170.195,47.458,159.114
C02554=1025.713,266.393,374.576,170.191,47.460,159.114
C02555=1025.705,266.145,374.606,170.188,47.463,159.114
C02556=1025.700,265.896,374.636,170.183,47.465,159.114
C02557=1025.693,265.648,374.666,170.180,47.467,159.114
C02558=1025.686,265.400,374.695,170.175,47.469,159.114
C02559=1025.680,265.152,374.725,170.172,47.471,159.114
C02560=1025.673,264.904,374.755,170.167,47.474,159.113
C02561=1025.667,264.656,374.784,170.163,47.476,159.114
C02562=1025.660,264.408,374.815,170.160,47.478,159.113
C02563=1025.654,264.159,374.844,170.155,47.480,159.113
C02564=1025.643,263.760,374.892,170.149,47.484,159.113
C02565=1025.632,263.361,374.939,170.143,47.488,159.113
C02566=1025.622,262.962,374.987,170.137,47.491,159.113
C02567=1025.612,262.564,375.034,170.130,47.495,159.113
C02568=1025.604,262.315,375.064,170.126,47.497,159.113
C02569=1025.599,262.067,375.094,170.122,47.500,159.113
C02570=1025.593,261.819,375.123,170.119,47.502,159.113
C02571=1025.586,261.571,375.153,170.114,47.504,159.113
C02572=1025.579,261.323,375.182,170.110,47.506,159.113
C02573=1025.573,261.075,375.212,170.106,47.509,159.113
C02574=1025.566,260.826,375.241,170.103,47.511,159.113
C02575=1025.560,260.578,375.270,170.099,47.513,159.113
C02576=1025.552,260.330,375.300,170.094,47.516,159.113
C02577=1025.546,260.082,375.330,170.091,47.518,159.113
C02578=1025.540,259.834,375.359,170.087,47.521,159.113
C02579=1025.532,259.585,375.387,170.083,47.523,159.113
C02580=1025.526,259.337,375.416,170.079,47.526,159.113
C02581=1025.520,259.089,375.445,170.075,47.528,159.113
C02582=1025.513,258.841,375.476,170.072,47.530,159.113
C02583=1025.506,258.593,375.504,170.067,47.533,159.113
C02584=1025.499,258.345,375.533,170.064,47.535,159.113
C02585=1025.493,258.096,375.562,170.059,47.538,159.113
C02586=1025.486,257.848,375.592,170.056,47.540,159.114
C02587=1025.479,257.600,375.620,170.052,47.543,159.114
C02588=1025.473,257.351,375.649,170.048,47.545,159.114
C02589=1025.466,257.103,375.678,170.044,47.548,159.114
C02590=1025.460,256.855,375.707,170.040,47.550,159.114
C02591=1025.452,256.606,375.736,170.037,47.553,159.114
C02592=1025.446,256.358,375.765,170.032,47.555,159.114
C02593=1025.440,256.110,375.794,170.029,47.558,159.114
C02594=1025.434,255.862,375.823,170.025,47.561,159.114
C02595=1025.426,255.613,375.852,170.021,47.563,159.114
C02596=1025.420,255.365,375.881,170.018,47.565,159.114
C02597=1025.414,255.117,375.910,170.013,47.568,159.114
C02598=1025.407,254.869,375.939,170.010,47.571,159.114
C02599=1025.400,254.620,375.968,170.006,47.573,159.114
C02600=1025.394,254.372,375.997,170.002,47.576,159.114
C02601=1025.387,254.124,376.026,169.999,47.578,159.114
C02602=1025.381,253.876,376.055,169.994,47.581,159.114
C02603=1025.374,253.628,376.084,169.991,47.583,159.114
C02604=1025.367,253.379,376.113,169.986,47.586,159.114
C02605=1025.361,253.131,376.142,169.983,47.588,159.114
C02606=1025.355,252.883,376.171,169.980,47.591,159.114
C02607=1025.348,252.635,376.200,169.975,47.593,159.115
C02608=1025.342,252.386,376.228,169.972,47.596,159.115
C02609=1025.335,252.138,376.257,169.967,47.599,159.115
C02610=1025.329,251.890,376.286,169.964,47.601,159.115
C02611=1025.322,251.642,376.315,169.961,47.603,159.115
C02612=1025.315,251.394,376.344,169.956,47.606,159.115
C02613=1025.309,251.145,376.372,169.953,47.609,159.115
C02614=1025.302,250.897,376.401,169.949,47.611,159.115
C02615=1025.296,250.649,376.430,169.945,47.614,159.115
C02616=1025.290,250.401,376.459,169.942,47.617,159.115
C02617=1025.283,250.152,376.488,169.937,47.619,159.115
C02618=1025.276,249.903,376.516,169.934,47.622,159.115
C02619=1025.270,249.655,376.545,169.931,47.624,159.115
C02620=1025.260,249.255,376.591,169.925,47.629,159.116
C02621=1025.250,248.855,376.638,169.919,47.633,159.116
C02622=1025.240,248.454,376.684,169.913,47.637,159.116
C02623=1025.228,248.053,376.730,169.907,47.641,159.116
C02624=1025.223,247.805,376.758,169.902,47.644,159.116
C02625=1025.216,247.557,376.787,169.899,47.647,159.116
C02626=1025.210,247.308,376.816,169.896,47.649,159.116
C02627=1025.203,247.060,376.844,169.891,47.652,159.116
C02628=1025.197,246.812,376.873,169.888,47.655,159.116
C02629=1025.191,246.564,376.902,169.885,47.657,159.116
C02630=1025.184,246.315,376.930,169.880,47.660,159.116
C02631=1025.178,246.067,376.959,169.877,47.663,159.117
C02632=1025.172,245.818,376.987,169.874,47.665,159.117
C02633=1025.166,245.570,377.016,169.869,47.668,159.117
C02634=1025.159,245.322,377.044,169.866,47.671,159.117
C02635=1025.153,245.074,377.073,169.863,47.673,159.117
C02636=1025.147,244.826,377.102,169.858,47.676,159.117
C02637=1025.140,244.577,377.130,169.855,47.679,159.117
C02638=1025.134,244.329,377.159,169.852,47.682,159.117
C02639=1025.128,244.081,377.187,169.847,47.684,159.117
C02640=1025.122,243.833,377.216,169.844,47.687,159.117
C02641=1025.115,243.584,377.244,169.841,47.690,159.118
C02642=1025.109,243.336,377.271,169.836,47.693,159.118
C02643=1025.102,243.088,377.300,169.833,47.696,159.118
C02644=1025.096,242.839,377.328,169.830,47.698,159.118
C02645=1025.090,242.591,377.356,169.825,47.701,159.118
C02646=1025.083,242.343,377.385,169.822,47.704,159.118
C02647=1025.077,242.094,377.413,169.819,47.706,159.118
C02648=1025.070,241.846,377.441,169.815,47.710,159.118
C02649=1025.063,241.598,377.469,169.811,47.712,159.119
C02650=1025.057,241.349,377.498,169.808,47.715,159.119
C02651=1025.051,241.101,377.525,169.804,47.718,159.119
C02652=1025.045,240.852,377.554,169.801,47.721,159.119
C02653=1025.038,240.605,377.582,169.797,47.723,159.119
C02654=1025.032,240.356,377.610,169.793,47.727,159.119
C02655=1025.026,240.107,377.638,169.790,47.729,159.119
C02656=1025.019,239.859,377.666,169.787,47.732,159.120
C02657=1025.013,239.610,377.694,169.782,47.735,159.120
C02658=1025.006,239.362,377.722,169.779,47.738,159.120
C02659=1024.999,239.114,377.750,169.775,47.742,159.120
C02660=1024.993,238.866,377.778,169.772,47.744,159.120
C02661=1024.986,238.617,377.806,169.769,47.747,159.120
C02662=1024.980,238.369,377.833,169.765,47.750,159.121
C02663=1024.974,238.121,377.861,169.761,47.753,159.121
C02664=1024.967,237.872,377.889,169.758,47.756,159.121
C02665=1024.961,237.624,377.917,169.754,47.759,159.121
C02666=1024.954,237.375,377.944,169.751,47.762,159.121
C02667=1024.947,237.127,377.972,169.747,47.765,159.121
C02668=1024.941,236.878,378.000,169.743,47.768,159.122
C02669=1024.935,236.630,378.028,169.740,47.771,159.122
C02670=1024.929,236.382,378.056,169.736,47.774,159.122
C02671=1024.922,236.133,378.083,169.733,47.777,159.122
C02672=1024.915,235.885,378.111,169.730,47.780,159.122
C02673=1024.908,235.637,378.139,169.725,47.783,159.122
C02674=1024.902,235.388,378.166,169.722,47.786,159.123
C02675=1024.896,235.140,378.194,169.718,47.789,159.123
C02676=1024.885,234.733,378.239,169.713,47.795,159.123
C02677=1024.875,234.326,378.284,169.707,47.799,159.123
C02678=1024.864,233.919,378.330,169.701,47.805,159.124
C02679=1024.853,233.513,378.374,169.696,47.809,159.124
C02680=1024.847,233.264,378.402,169.692,47.812,159.124
C02681=1024.841,233.016,378.431,169.688,47.816,159.124
C02682=1024.835,232.767,378.457,169.685,47.819,159.125
C02683=1024.828,232.519,378.485,169.682,47.822,159.125
C02684=1024.822,232.270,378.513,169.678,47.825,159.125
C02685=1024.815,232.022,378.540,169.675,47.828,159.125
C02686=1024.809,231.774,378.568,169.671,47.831,159.125
C02687=1024.802,231.525,378.595,169.668,47.834,159.126
C02688=1024.796,231.277,378.622,169.664,47.837,159.126
C02689=1024.790,231.029,378.650,169.660,47.841,159.126
C02690=1024.783,230.781,378.678,169.657,47.844,159.126
C02691=1024.777,230.532,378.705,169.654,47.847,159.126
C02692=1024.770,230.283,378.732,169.650,47.850,159.127
C02693=1024.764,230.035,378.760,169.647,47.853,159.127
C02694=1024.757,229.786,378.787,169.644,47.856,159.127
C02695=1024.751,229.538,378.814,169.639,47.859,159.127
C02696=1024.745,229.290,378.842,169.636,47.862,159.127
C02697=1024.738,229.041,378.869,169.633,47.865,159.128
C02698=1024.732,228.793,378.897,169.629,47.869,159.128
C02699=1024.726,228.544,378.923,169.626,47.872,159.128
C02700=1024.719,228.296,378.951,169.623,47.875,159.128
C02701=1024.713,228.047,378.978,169.619,47.878,159.128
C02702=1024.707,227.799,379.005,169.616,47.881,159.129
C02703=1024.699,227.551,379.032,169.613,47.885,159.129
C02704=1024.693,227.302,379.059,169.609,47.889,159.129
C02705=1024.687,227.054,379.087,169.606,47.892,159.130
C02706=1024.681,226.805,379.114,169.602,47.895,159.130
C02707=1024.674,226.557,379.142,169.599,47.898,159.130
C02708=1024.667,226.309,379.168,169.596,47.901,159.130
C02709=1024.661,226.059,379.195,169.592,47.905,159.130
C02710=1024.654,225.811,379.222,169.589,47.908,159.131
C02711=1024.648,225.563,379.248,169.585,47.912,159.131
C02712=1024.641,225.315,379.276,169.582,47.915,159.131
C02713=1024.635,225.066,379.303,169.579,47.918,159.131
C02714=1024.628,224.817,379.329,169.574,47.921,159.132
C02715=1024.622,224.569,379.357,169.571,47.925,159.132
C02716=1024.616,224.321,379.384,169.569,47.928,159.132
C02717=1024.609,224.072,379.410,169.565,47.932,159.132
C02718=1024.603,223.824,379.437,169.561,47.935,159.133
C02719=1024.596,223.575,379.464,169.557,47.938,159.133
C02720=1024.589,223.326,379.491,169.554,47.941,159.133
C02721=1024.583,223.078,379.517,169.552,47.945,159.134
C02722=1024.577,222.830,379.545,169.547,47.948,159.134
C02723=1024.571,222.581,379.572,169.544,47.952,159.134
C02724=1024.564,222.332,379.598,169.541,47.955,159.134
C02725=1024.558,222.085,379.626,169.538,47.959,159.135
C02726=1024.551,221.836,379.653,169.534,47.962,159.135
C02727=1024.544,221.587,379.679,169.531,47.965,159.135
C02728=1024.538,221.339,379.706,169.527,47.968,159.135
C02729=1024.532,221.090,379.733,169.525,47.972,159.136
C02730=1024.525,220.842,379.759,169.520,47.976,159.136
C02731=1024.519,220.593,379.786,169.517,47.979,159.136
C02732=1024.508,220.178,379.831,169.512,47.985,159.137
C02733=1024.498,219.764,379.875,169.507,47.990,159.137
C02734=1024.487,219.349,379.920,169.501,47.996,159.138
C02735=1024.476,218.935,379.965,169.495,48.002,159.138
C02736=1024.470,218.686,379.991,169.492,48.005,159.138
C02737=1024.463,218.438,380.018,169.488,48.009,159.139
C02738=1024.458,218.189,380.044,169.486,48.012,159.139
C02739=1024.450,217.941,380.071,169.481,48.016,159.139
C02740=1024.444,217.693,380.097,169.479,48.020,159.140
C02741=1024.438,217.443,380.124,169.476,48.023,159.140
C02742=1024.431,217.195,380.150,169.472,48.027,159.140
C02743=1024.425,216.946,380.177,169.469,48.030,159.140
C02744=1024.418,216.698,380.203,169.465,48.034,159.141
C02745=1024.411,216.450,380.229,169.462,48.037,159.141
C02746=1024.405,216.201,380.256,169.459,48.041,159.141
C02747=1024.398,215.952,380.282,169.455,48.044,159.142
C02748=1024.392,215.704,380.308,169.452,48.048,159.142
C02749=1024.385,215.455,380.335,169.448,48.052,159.142
C02750=1024.379,215.207,380.361,169.446,48.055,159.143
C02751=1024.373,214.959,380.388,169.443,48.059,159.143
C02752=1024.366,214.710,380.415,169.439,48.062,159.143
C02753=1024.360,214.462,380.440,169.436,48.066,159.144
C02754=1024.353,214.212,380.467,169.433,48.069,159.144
C02755=1024.347,213.964,380.493,169.429,48.073,159.144
C02756=1024.340,213.716,380.519,169.426,48.077,159.144
C02757=1024.334,213.467,380.546,169.422,48.081,159.145
C02758=1024.327,213.219,380.572,169.420,48.084,159.145
C02759=1024.321,212.970,380.599,169.416,48.088,159.145
C02760=1024.315,212.722,380.624,169.413,48.092,159.146
C02761=1024.308,212.473,380.650,169.410,48.095,159.146
C02762=1024.302,212.224,380.677,169.406,48.099,159.146
C02763=1024.295,211.976,380.704,169.403,48.103,159.147
C02764=1024.288,211.728,380.730,169.400,48.106,159.147
C02765=1024.283,211.479,380.756,169.396,48.110,159.147
C02766=1024.276,211.231,380.782,169.394,48.114,159.148
C02767=1024.270,210.981,380.809,169.390,48.117,159.148
C02768=1024.263,210.733,380.835,169.387,48.121,159.148
C02769=1024.257,210.485,380.860,169.384,48.125,159.149
C02770=1024.251,210.236,380.887,169.381,48.128,159.149
C02771=1024.244,209.988,380.913,169.377,48.132,159.149
C02772=1024.238,209.739,380.939,169.374,48.136,159.150
C02773=1024.231,209.490,380.965,169.371,48.140,159.150
C02774=1024.224,209.242,380.991,169.368,48.143,159.150
C02775=1024.218,208.994,381.017,169.364,48.147,159.151
C02776=1024.212,208.744,381.044,169.361,48.151,159.151
C02777=1024.206,208.496,381.069,169.358,48.155,159.152
C02778=1024.199,208.248,381.095,169.354,48.158,159.152
C02779=1024.193,208.000,381.121,169.352,48.162,159.152
C02780=1024.186,207.750,381.147,169.348,48.166,159.153
C02781=1024.179,207.502,381.173,169.345,48.170,159.153
C02782=1024.173,207.254,381.198,169.342,48.173,159.153
C02783=1024.167,207.005,381.225,169.339,48.178,159.154
C02784=1024.161,206.756,381.250,169.335,48.181,159.154
C02785=1024.154,206.508,381.277,169.332,48.185,159.154
C02786=1024.148,206.259,381.302,169.329,48.189,159.155
C02787=1024.141,206.010,381.328,169.326,48.192,159.155
C02788=1024.131,205.598,381.371,169.320,48.199,159.156
C02789=1024.119,205.186,381.413,169.315,48.205,159.156
C02790=1024.108,204.775,381.456,169.311,48.212,159.157
C02791=1024.098,204.363,381.499,169.304,48.218,159.158
C02792=1024.074,203.330,381.599,168.894,48.119,159.079
C02793=1024.068,203.082,381.624,168.891,48.124,159.080
C02794=1024.063,202.833,381.648,168.886,48.128,159.080
C02795=1024.057,202.584,381.672,168.882,48.133,159.080
C02796=1024.051,202.336,381.696,168.878,48.138,159.081
C02797=1024.046,202.087,381.721,168.873,48.142,159.081
C02798=1024.041,201.838,381.744,168.870,48.147,159.082
C02799=1024.034,201.589,381.768,168.865,48.152,159.082
C02800=1024.029,201.340,381.792,168.862,48.157,159.083
C02801=1024.024,201.092,381.817,168.857,48.161,159.083
C02802=1024.018,200.843,381.841,168.854,48.166,159.083
C02803=1024.012,200.594,381.865,168.849,48.171,159.084
C02804=1024.007,200.346,381.889,168.846,48.176,159.084
C02805=1024.001,200.097,381.913,168.841,48.180,159.084
C02806=1023.996,199.847,381.937,168.836,48.185,159.085
C02807=1023.990,199.599,381.961,168.833,48.190,159.085
C02808=1023.984,199.350,381.985,168.828,48.195,159.086
C02809=1023.978,199.101,382.009,168.825,48.200,159.086
C02810=1023.972,198.852,382.032,168.820,48.205,159.087
C02811=1023.967,198.604,382.056,168.816,48.210,159.087
C02812=1023.961,198.356,382.080,168.813,48.215,159.088
C02813=1023.955,198.106,382.104,168.808,48.220,159.088
C02814=1023.949,197.857,382.128,168.805,48.225,159.089
C02815=1023.943,197.608,382.151,168.800,48.230,159.089
C02816=1023.938,197.360,382.175,168.796,48.234,159.089
C02817=1023.931,197.111,382.199,168.792,48.239,159.090
C02818=1023.926,196.862,382.222,168.787,48.244,159.090
C02819=1023.920,196.613,382.246,168.784,48.249,159.091
C02820=1023.915,196.365,382.269,168.780,48.254,159.091
C02821=1023.909,196.116,382.293,168.776,48.259,159.091
C02822=1023.903,195.866,382.317,168.772,48.264,159.092
C02823=1023.898,195.618,382.341,168.768,48.268,159.092
C02824=1023.892,195.369,382.364,168.764,48.274,159.093
C02825=1023.886,195.121,382.388,168.760,48.278,159.093
C02826=1023.881,194.871,382.411,168.756,48.283,159.094
C02827=1023.875,194.623,382.435,168.751,48.288,159.094
C02828=1023.868,194.373,382.458,168.748,48.293,159.095
C02829=1023.863,194.125,382.482,168.743,48.298,159.095
C02830=1023.857,193.876,382.505,168.740,48.303,159.096
C02831=1023.852,193.627,382.529,168.736,48.308,159.096
C02832=1023.846,193.379,382.552,168.732,48.313,159.096
C02833=1023.840,193.130,382.576,168.728,48.318,159.097
C02834=1023.835,192.881,382.600,168.724,48.323,159.097
C02835=1023.830,192.632,382.623,168.720,48.328,159.098
C02836=1023.824,192.384,382.647,168.716,48.333,159.098
C02837=1023.819,192.135,382.670,168.713,48.338,159.099
C02838=1023.812,191.886,382.694,168.708,48.343,159.099
C02839=1023.807,191.636,382.717,168.705,48.347,159.100
C02840=1023.801,191.388,382.740,168.701,48.353,159.100
C02841=1023.795,191.139,382.764,168.697,48.357,159.101
C02842=1023.790,190.890,382.787,168.693,48.362,159.101
C02843=1023.784,190.641,382.810,168.689,48.367,159.101
C02844=1023.778,190.393,382.834,168.685,48.372,159.102
C02845=1023.773,190.144,382.858,168.681,48.377,159.102
C02846=1023.768,189.895,382.881,168.677,48.382,159.103
C02847=1023.762,189.646,382.905,168.673,48.387,159.103
C02848=1023.757,189.397,382.928,168.670,48.392,159.104
C02849=1023.751,189.148,382.951,168.666,48.397,159.104
C02850=1023.746,188.899,382.974,168.662,48.402,159.105
C02851=1023.740,188.651,382.998,168.658,48.407,159.105
C02852=1023.734,188.402,383.021,168.654,48.412,159.106
C02853=1023.729,188.120,383.048,168.650,48.417,159.106
C02854=1023.722,187.837,383.074,168.646,48.423,159.107
C02855=1023.716,187.555,383.100,168.642,48.428,159.107
C02856=1023.709,187.273,383.127,168.636,48.434,159.108
C02857=1023.704,187.024,383.150,168.633,48.439,159.108
C02858=1023.699,186.775,383.173,168.630,48.444,159.109
C02859=1023.693,186.526,383.196,168.625,48.449,159.109
C02860=1023.688,186.277,383.220,168.622,48.454,159.110
C02861=1023.682,186.029,383.243,168.618,48.459,159.110
C02862=1023.676,185.780,383.266,168.614,48.464,159.110
C02863=1023.671,185.531,383.290,168.610,48.469,159.111
C02864=1023.666,185.283,383.312,168.607,48.473,159.111
C02865=1023.660,185.034,383.335,168.602,48.479,159.112
C02866=1023.655,184.784,383.359,168.599,48.484,159.113
C02867=1023.650,184.536,383.382,168.596,48.489,159.113
C02868=1023.644,184.287,383.405,168.592,48.494,159.113
C02869=1023.639,184.037,383.428,168.588,48.499,159.114
C02870=1023.633,183.789,383.451,168.585,48.504,159.114
C02871=1023.627,183.540,383.475,168.580,48.509,159.115
C02872=1023.623,183.292,383.498,168.577,48.514,159.115
C02873=1023.617,183.043,383.521,168.573,48.518,159.116
C02874=1023.612,182.793,383.543,168.569,48.523,159.116
C02875=1023.607,182.544,383.567,168.566,48.528,159.117
C02876=1023.601,182.295,383.590,168.562,48.533,159.117
C02877=1023.595,182.046,383.613,168.558,48.539,159.118
C02878=1023.589,181.798,383.635,168.555,48.544,159.118
C02879=1023.583,181.548,383.657,168.550,48.549,159.119
C02880=1023.578,181.299,383.680,168.547,48.554,159.119
C02881=1023.572,181.050,383.703,168.543,48.559,159.120
C02882=1023.566,180.803,383.725,168.539,48.564,159.120
C02883=1023.561,180.553,383.747,168.536,48.570,159.121
C02884=1023.555,180.304,383.770,168.532,48.575,159.121
C02885=1023.548,180.056,383.793,168.529,48.580,159.122
C02886=1023.543,179.806,383.815,168.524,48.586,159.122
C02887=1023.537,179.557,383.838,168.521,48.590,159.123
C02888=1023.531,179.308,383.861,168.518,48.596,159.123
C02889=1023.526,179.060,383.882,168.513,48.601,159.124
C02890=1023.520,178.811,383.905,168.510,48.607,159.125
C02891=1023.515,178.561,383.927,168.506,48.612,159.125
C02892=1023.508,178.313,383.950,168.502,48.616,159.125
C02893=1023.503,178.064,383.972,168.499,48.622,159.126
C02894=1023.497,177.814,383.995,168.495,48.627,159.127
C02895=1023.492,177.566,384.017,168.492,48.633,159.127
C02896=1023.486,177.317,384.039,168.488,48.638,159.128
C02897=1023.480,177.068,384.062,168.484,48.643,159.128
C02898=1023.474,176.819,384.085,168.481,48.648,159.129
C02899=1023.468,176.570,384.106,168.476,48.653,159.129
C02900=1023.463,176.322,384.129,168.473,48.659,159.130
C02901=1023.458,176.072,384.151,168.470,48.664,159.130
C02902=1023.452,175.823,384.174,168.465,48.669,159.131
C02903=1023.446,175.574,384.196,168.462,48.674,159.131
C02904=1023.441,175.326,384.218,168.459,48.679,159.132
C02905=1023.435,175.076,384.241,168.455,48.685,159.132
C02906=1023.429,174.828,384.263,168.451,48.690,159.133
C02907=1023.423,174.578,384.285,168.448,48.695,159.133
C02908=1023.418,174.330,384.308,168.444,48.700,159.134
C02909=1023.412,174.081,384.329,168.441,48.705,159.134
C02910=1023.407,173.831,384.352,168.438,48.711,159.135
C02911=1023.401,173.583,384.374,168.434,48.716,159.136
C02912=1023.396,173.334,384.397,168.430,48.721,159.136
C02913=1023.390,173.085,384.419,168.427,48.726,159.137
C02914=1023.385,172.836,384.441,168.423,48.731,159.137
C02915=1023.379,172.587,384.463,168.419,48.737,159.138
C02916=1023.373,172.338,384.485,168.416,48.742,159.138
C02917=1023.367,172.055,384.510,168.412,48.748,159.139
C02918=1023.360,171.773,384.535,168.408,48.754,159.139
C02919=1023.354,171.491,384.561,168.403,48.759,159.140
C02920=1023.348,171.207,384.586,168.400,48.766,159.141
C02921=1023.342,170.959,384.608,168.396,48.771,159.141
C02922=1023.337,170.710,384.631,168.393,48.776,159.142
C02923=1023.332,170.461,384.652,168.389,48.781,159.142
C02924=1023.326,170.212,384.675,168.385,48.786,159.143
C02925=1023.320,169.963,384.697,168.382,48.792,159.143
C02926=1023.315,169.714,384.719,168.379,48.797,159.144
C02927=1023.309,169.465,384.740,168.375,48.802,159.144
C02928=1023.303,169.216,384.763,168.372,48.807,159.145
C02929=1023.299,168.967,384.785,168.368,48.812,159.145
C02930=1023.292,168.718,384.807,168.365,48.818,159.146
C02931=1023.287,168.469,384.829,168.362,48.823,159.147
C02932=1023.282,168.220,384.852,168.358,48.829,159.147
C02933=1023.276,167.971,384.873,168.354,48.833,159.148
C02934=1023.271,167.722,384.895,168.351,48.838,159.148
C02935=1023.265,167.472,384.917,168.348,48.844,159.149
C02936=1023.260,167.225,384.939,168.344,48.849,159.149
C02937=1023.254,166.975,384.962,168.340,48.855,159.150
C02938=1023.249,166.726,384.984,168.337,48.859,159.150
C02939=1023.243,166.477,385.005,168.334,48.864,159.151
C02940=1023.238,166.228,385.027,168.330,48.870,159.151
C02941=1023.233,165.979,385.050,168.327,48.875,159.152
C02942=1023.227,165.731,385.071,168.324,48.880,159.153
C02943=1023.222,165.481,385.093,168.320,48.885,159.153
C02944=1023.217,165.232,385.115,168.316,48.890,159.153
C02945=1023.211,164.983,385.137,168.313,48.896,159.154
C02946=1023.206,164.734,385.159,168.310,48.901,159.155
C02947=1023.200,164.485,385.181,168.307,48.906,159.155
C02948=1023.195,164.237,385.203,168.303,48.911,159.156
C02949=1023.189,163.987,385.225,168.299,48.916,159.156
C02950=1023.184,163.739,385.247,168.296,48.922,159.157
C02951=1023.178,163.489,385.269,168.293,48.927,159.157
C02952=1023.173,163.241,385.291,168.289,48.932,159.158
C02953=1023.168,162.991,385.313,168.286,48.937,159.158
C02954=1023.162,162.743,385.334,168.283,48.942,159.159
C02955=1023.157,162.494,385.356,168.280,48.948,159.160
C02956=1023.152,162.244,385.378,168.276,48.953,159.160
C02957=1023.146,161.996,385.399,168.273,48.958,159.161
C02958=1023.141,161.746,385.422,168.269,48.963,159.161
C02959=1023.136,161.497,385.444,168.265,48.968,159.162
C02960=1023.130,161.248,385.465,168.262,48.974,159.162
C02961=1023.125,160.999,385.487,168.259,48.979,159.163
C02962=1023.120,160.751,385.508,168.256,48.984,159.163
C02963=1023.114,160.501,385.531,168.253,48.989,159.164
C02964=1023.109,160.253,385.552,168.249,48.994,159.164
C02965=1023.103,160.003,385.574,168.246,49.000,159.165
C02966=1023.098,159.755,385.596,168.243,49.005,159.165
C02967=1023.094,159.506,385.618,168.240,49.010,159.166
C02968=1023.087,159.257,385.639,168.236,49.015,159.167
C02969=1023.083,159.008,385.661,168.233,49.020,159.167
C02970=1023.076,158.759,385.683,168.229,49.026,159.168
C02971=1023.071,158.509,385.703,168.226,49.031,159.168
C02972=1023.066,158.261,385.725,168.223,49.036,159.169
C02973=1023.060,158.011,385.747,168.220,49.042,159.169
C02974=1023.055,157.763,385.768,168.217,49.047,159.170
C02975=1023.049,157.513,385.789,168.213,49.052,159.171
C02976=1023.043,157.265,385.810,168.209,49.058,159.171
C02977=1023.038,157.016,385.832,168.206,49.064,159.172
C02978=1023.033,156.766,385.853,168.203,49.069,159.172
C02979=1023.027,156.517,385.875,168.200,49.074,159.173
C02980=1023.021,156.269,385.896,168.196,49.079,159.173
C02981=1023.015,155.985,385.920,168.193,49.086,159.174
C02982=1023.008,155.702,385.944,168.189,49.092,159.175
C02983=1023.002,155.419,385.968,168.185,49.098,159.176
C02984=1022.996,155.136,385.992,168.181,49.104,159.176
C02985=1022.991,154.887,386.014,168.178,49.110,159.177
C02986=1022.986,154.638,386.035,168.174,49.115,159.177
C02987=1022.980,154.389,386.056,168.171,49.120,159.178
C02988=1022.974,154.140,386.077,168.168,49.125,159.178
C02989=1022.969,153.891,386.098,168.165,49.131,159.179
C02990=1022.963,153.642,386.120,168.162,49.136,159.180
C02991=1022.958,153.393,386.141,168.159,49.141,159.180
C02992=1022.952,153.144,386.162,168.156,49.147,159.181
C02993=1022.947,152.894,386.183,168.153,49.152,159.181
C02994=1022.941,152.646,386.204,168.148,49.158,159.182
C02995=1022.936,152.397,386.225,168.145,49.163,159.183
C02996=1022.930,152.148,386.246,168.142,49.169,159.183
C02997=1022.924,151.898,386.267,168.139,49.174,159.184
C02998=1022.919,151.650,386.288,168.136,49.179,159.184
C02999=1022.914,151.401,386.309,168.133,49.185,159.185
C03000=1022.907,151.152,386.330,168.129,49.190,159.185
C03001=1022.902,150.902,386.351,168.126,49.195,159.186
C03002=1022.897,150.654,386.372,168.123,49.201,159.187
C03003=1022.891,150.404,386.393,168.119,49.206,159.187
C03004=1022.885,150.155,386.414,168.116,49.212,159.188
C03005=1022.880,149.906,386.435,168.113,49.218,159.188
C03006=1022.875,149.657,386.456,168.110,49.222,159.189
C03007=1022.868,149.408,386.477,168.107,49.228,159.190
C03008=1022.863,149.159,386.498,168.104,49.234,159.190
C03009=1022.858,148.910,386.518,168.100,49.239,159.191
C03010=1022.852,148.661,386.540,168.097,49.244,159.191
C03011=1022.847,148.412,386.560,168.094,49.250,159.192
C03012=1022.841,148.162,386.581,168.091,49.255,159.193
C03013=1022.836,147.914,386.602,168.088,49.260,159.193
C03014=1022.830,147.665,386.623,168.085,49.266,159.194
C03015=1022.825,147.416,386.643,168.082,49.272,159.194
C03016=1022.819,147.167,386.665,168.079,49.276,159.195
C03017=1022.814,146.917,386.686,168.076,49.282,159.196
C03018=1022.809,146.668,386.706,168.071,49.288,159.196
C03019=1022.803,146.419,386.727,168.068,49.293,159.197
C03020=1022.798,146.171,386.748,168.065,49.299,159.197
C03021=1022.792,145.921,386.769,168.062,49.304,159.198
C03022=1022.787,145.672,386.789,168.059,49.310,159.199
C03023=1022.781,145.423,386.809,168.056,49.315,159.199
C03024=1022.775,145.174,386.830,168.053,49.320,159.200
C03025=1022.770,144.925,386.851,168.050,49.326,159.200
C03026=1022.764,144.675,386.872,168.047,49.332,159.201
C03027=1022.758,144.427,386.892,168.044,49.337,159.202
C03028=1022.753,144.177,386.913,168.040,49.342,159.202
C03029=1022.747,143.928,386.933,168.037,49.348,159.203
C03030=1022.742,143.679,386.954,168.034,49.353,159.203
C03031=1022.736,143.430,386.974,168.031,49.359,159.204
C03032=1022.730,143.181,386.995,168.027,49.365,159.205
C03033=1022.725,142.932,387.016,168.024,49.370,159.205
C03034=1022.720,142.683,387.036,168.021,49.376,159.206
C03035=1022.714,142.434,387.056,168.018,49.381,159.206
C03036=1022.708,142.185,387.077,168.015,49.387,159.207
C03037=1022.703,141.936,387.098,168.012,49.392,159.208
C03038=1022.698,141.687,387.118,168.009,49.397,159.208
C03039=1022.691,141.437,387.138,168.006,49.403,159.209
C03040=1022.686,141.188,387.159,168.003,49.409,159.210
C03041=1022.681,140.939,387.180,168.000,49.414,159.210
C03042=1022.675,140.690,387.200,167.997,49.419,159.211
C03043=1022.669,140.441,387.220,167.994,49.425,159.211
C03044=1022.664,140.192,387.241,167.991,49.431,159.212
C03045=1022.658,139.909,387.264,167.987,49.436,159.213
C03046=1022.651,139.626,387.287,167.984,49.443,159.213
C03047=1022.645,139.342,387.310,167.980,49.449,159.214
C03048=1022.639,139.058,387.334,167.976,49.455,159.215
C03049=1022.633,138.809,387.354,167.973,49.461,159.215
C03050=1022.628,138.560,387.374,167.970,49.466,159.216
C03051=1022.623,138.311,387.395,167.967,49.472,159.217
C03052=1022.617,138.062,387.415,167.964,49.477,159.217
C03053=1022.611,137.813,387.435,167.961,49.483,159.218
C03054=1022.606,137.564,387.456,167.958,49.489,159.218
C03055=1022.601,137.315,387.475,167.955,49.494,159.219
C03056=1022.595,137.066,387.496,167.952,49.499,159.220
C03057=1022.589,136.817,387.516,167.949,49.505,159.220
C03058=1022.584,136.568,387.536,167.946,49.510,159.221
C03059=1022.578,136.319,387.556,167.943,49.516,159.222
C03060=1022.573,136.070,387.577,167.940,49.522,159.222
C03061=1022.568,135.820,387.597,167.937,49.527,159.223
C03062=1022.562,135.571,387.617,167.934,49.532,159.223
C03063=1022.557,135.322,387.637,167.931,49.538,159.224
C03064=1022.551,135.073,387.657,167.928,49.544,159.225
C03065=1022.544,134.824,387.677,167.925,49.549,159.225
C03066=1022.539,134.574,387.697,167.922,49.555,159.226
C03067=1022.533,134.325,387.717,167.918,49.560,159.226
C03068=1022.528,134.076,387.738,167.915,49.566,159.227
C03069=1022.522,133.827,387.757,167.912,49.571,159.228
C03070=1022.517,133.577,387.778,167.909,49.577,159.228
C03071=1022.511,133.329,387.798,167.906,49.583,159.229
C03072=1022.506,133.080,387.818,167.904,49.588,159.230
C03073=1022.501,132.831,387.837,167.901,49.594,159.230
C03074=1022.495,132.582,387.858,167.897,49.599,159.231
C03075=1022.489,132.333,387.877,167.894,49.605,159.231
C03076=1022.484,132.083,387.897,167.891,49.610,159.232
C03077=1022.478,131.834,387.917,167.888,49.616,159.233
C03078=1022.473,131.585,387.938,167.885,49.622,159.233
C03079=1022.467,131.336,387.957,167.882,49.627,159.234
C03080=1022.462,131.087,387.978,167.879,49.632,159.235
C03081=1022.456,130.838,387.998,167.876,49.638,159.235
C03082=1022.451,130.588,388.017,167.874,49.643,159.236
C03083=1022.445,130.339,388.037,167.871,49.649,159.237
C03084=1022.439,130.090,388.057,167.868,49.655,159.237
C03085=1022.434,129.841,388.077,167.865,49.660,159.238
C03086=1022.429,129.591,388.096,167.862,49.665,159.238
C03087=1022.423,129.342,388.116,167.859,49.671,159.239
C03088=1022.417,129.093,388.136,167.856,49.677,159.240
C03089=1022.411,128.844,388.156,167.852,49.683,159.240
C03090=1022.405,128.595,388.175,167.849,49.688,159.241
C03091=1022.399,128.346,388.195,167.846,49.694,159.242
C03092=1022.394,128.096,388.215,167.843,49.700,159.242
C03093=1022.388,127.847,388.235,167.840,49.705,159.243
C03094=1022.383,127.599,388.253,167.837,49.711,159.243
C03095=1022.377,127.349,388.273,167.834,49.717,159.244
C03096=1022.371,127.100,388.293,167.831,49.722,159.245
C03097=1022.366,126.851,388.312,167.829,49.728,159.245
C03098=1022.360,126.602,388.332,167.826,49.734,159.246
C03099=1022.355,126.352,388.352,167.823,49.739,159.247
C03100=1022.349,126.103,388.371,167.820,49.745,159.247
C03101=1022.343,125.854,388.391,167.817,49.751,159.248
C03102=1022.337,125.605,388.410,167.814,49.756,159.249
C03103=1022.332,125.355,388.429,167.811,49.762,159.249
C03104=1022.326,125.107,388.449,167.808,49.768,159.250
C03105=1022.321,124.858,388.468,167.805,49.773,159.251
C03106=1022.315,124.608,388.487,167.802,49.779,159.251
C03107=1022.310,124.359,388.508,167.799,49.785,159.252
C03108=1022.304,124.110,388.527,167.797,49.790,159.253
C03109=1022.298,123.826,388.550,167.794,49.797,159.253
C03110=1022.291,123.544,388.571,167.790,49.803,159.254
C03111=1022.284,123.260,388.593,167.787,49.809,159.255
C03112=1022.278,122.977,388.615,167.783,49.816,159.256
C03113=1022.273,122.728,388.634,167.780,49.822,159.256
C03114=1022.267,122.478,388.655,167.778,49.827,159.257
C03115=1022.262,122.229,388.674,167.774,49.832,159.257
C03116=1022.256,121.980,388.694,167.771,49.838,159.258
C03117=1022.251,121.731,388.712,167.768,49.844,159.259
C03118=1022.245,121.482,388.732,167.765,49.849,159.259
C03119=1022.239,121.233,388.752,167.763,49.855,159.260
C03120=1022.234,120.983,388.771,167.760,49.861,159.261
C03121=1022.228,120.734,388.790,167.758,49.866,159.261
C03122=1022.223,120.485,388.809,167.755,49.872,159.262
C03123=1022.218,120.236,388.830,167.752,49.878,159.263
C03124=1022.212,119.986,388.849,167.749,49.883,159.263
C03125=1022.206,119.737,388.868,167.746,49.888,159.264
C03126=1022.200,119.488,388.887,167.743,49.894,159.264
C03127=1022.195,119.239,388.906,167.740,49.900,159.265
C03128=1022.189,118.990,388.926,167.737,49.905,159.266
C03129=1022.184,118.741,388.945,167.734,49.911,159.266
C03130=1022.178,118.491,388.965,167.731,49.917,159.267
C03131=1022.173,118.242,388.983,167.728,49.923,159.268
C03132=1022.167,117.993,389.003,167.726,49.928,159.268
C03133=1022.162,117.743,389.023,167.723,49.933,159.269
C03134=1022.156,117.494,389.042,167.720,49.939,159.270
C03135=1022.151,117.246,389.061,167.717,49.944,159.270
C03136=1022.146,116.996,389.081,167.714,49.950,159.271
C03137=1022.140,116.747,389.100,167.711,49.956,159.272
C03138=1022.134,116.497,389.119,167.708,49.962,159.272
C03139=1022.129,116.249,389.138,167.705,49.967,159.273
C03140=1022.123,115.999,389.157,167.703,49.972,159.273
C03141=1022.118,115.750,389.176,167.700,49.978,159.274
C03142=1022.113,115.501,389.195,167.697,49.983,159.275
C03143=1022.107,115.252,389.216,167.694,49.989,159.275
C03144=1022.102,115.002,389.235,167.691,49.995,159.276
C03145=1022.097,114.754,389.254,167.688,50.000,159.276
C03146=1022.091,114.504,389.273,167.685,50.006,159.277
C03147=1022.085,114.255,389.292,167.683,50.011,159.278
C03148=1022.080,114.006,389.311,167.680,50.017,159.278
C03149=1022.074,113.757,389.331,167.677,50.022,159.279
C03150=1022.069,113.507,389.350,167.675,50.028,159.280
C03151=1022.064,113.259,389.369,167.671,50.033,159.280
C03152=1022.058,113.009,389.388,167.668,50.039,159.281
C03153=1022.052,112.760,389.407,167.666,50.044,159.282
C03154=1022.048,112.511,389.427,167.664,50.050,159.282
C03155=1022.042,112.262,389.445,167.661,50.056,159.283
C03156=1022.036,112.012,389.465,167.658,50.061,159.284
C03157=1022.031,111.763,389.483,167.655,50.067,159.284
C03158=1022.025,111.513,389.502,167.652,50.072,159.285
C03159=1022.020,111.264,389.521,167.649,50.078,159.285
C03160=1022.014,111.015,389.540,167.646,50.084,159.286
C03161=1022.008,110.766,389.559,167.644,50.089,159.287
C03162=1022.002,110.517,389.578,167.641,50.095,159.287
C03163=1021.997,110.268,389.597,167.638,50.101,159.288
C03164=1021.992,110.018,389.615,167.635,50.106,159.289
C03165=1021.986,109.769,389.634,167.632,50.112,159.289
C03166=1021.980,109.520,389.653,167.629,50.118,159.290
C03167=1021.975,109.271,389.672,167.626,50.124,159.291
C03168=1021.969,109.021,389.690,167.624,50.129,159.291
C03169=1021.964,108.772,389.709,167.621,50.135,159.292
C03170=1021.958,108.523,389.728,167.618,50.141,159.293
C03171=1021.951,108.273,389.747,167.616,50.146,159.293
C03172=1021.946,107.992,389.768,167.612,50.153,159.294
C03173=1021.940,107.716,389.789,167.609,50.159,159.295
C03174=1021.933,107.441,389.809,167.606,50.165,159.295
C03175=1021.927,107.166,389.830,167.603,50.172,159.296
C03176=1021.920,106.890,389.850,167.599,50.178,159.297
C03177=1021.915,106.641,389.869,167.597,50.184,159.297
C03178=1021.910,106.392,389.888,167.595,50.189,159.298
C03179=1021.904,106.143,389.905,167.592,50.195,159.299
C03180=1021.898,105.893,389.925,167.589,50.201,159.300
C03181=1021.892,105.644,389.943,167.586,50.206,159.300
C03182=1021.887,105.395,389.961,167.583,50.212,159.301
C03183=1021.882,105.145,389.981,167.580,50.218,159.301
C03184=1021.876,104.897,389.999,167.577,50.224,159.302
C03185=1021.870,104.647,390.017,167.574,50.229,159.303
C03186=1021.864,104.399,390.036,167.573,50.235,159.304
C03187=1021.859,104.149,390.054,167.570,50.240,159.304
C03188=1021.854,103.900,390.073,167.567,50.246,159.305
C03189=1021.848,103.651,390.092,167.564,50.252,159.305
C03190=1021.842,103.401,390.110,167.561,50.258,159.306
C03191=1021.837,103.152,390.129,167.558,50.264,159.307
C03192=1021.831,102.902,390.147,167.555,50.269,159.307
C03193=1021.826,102.653,390.166,167.553,50.274,159.308
C03194=1021.820,102.404,390.184,167.550,50.280,159.309
C03195=1021.815,102.155,390.203,167.547,50.286,159.309
C03196=1021.809,101.906,390.222,167.544,50.291,159.310
C03197=1021.804,101.656,390.240,167.542,50.297,159.311
C03198=1021.798,101.407,390.259,167.539,50.303,159.311
C03199=1021.792,101.158,390.276,167.537,50.308,159.312
C03200=1021.787,100.909,390.296,167.534,50.314,159.313
C03201=1021.782,100.659,390.314,167.531,50.320,159.313
C03202=1021.775,100.410,390.333,167.528,50.325,159.314
C03203=1021.771,100.161,390.351,167.525,50.331,159.314
C03204=1021.764,99.912,390.369,167.522,50.336,159.315
C03205=1021.759,99.662,390.387,167.520,50.342,159.316
C03206=1021.754,99.413,390.407,167.517,50.348,159.316
C03207=1021.748,99.164,390.424,167.514,50.353,159.317
C03208=1021.742,98.914,390.442,167.512,50.359,159.318
C03209=1021.737,98.665,390.461,167.509,50.365,159.318
C03210=1021.731,98.416,390.479,167.506,50.371,159.319
C03211=1021.725,98.167,390.497,167.503,50.376,159.320
C03212=1021.719,97.917,390.515,167.500,50.382,159.320
C03213=1021.714,97.668,390.533,167.498,50.388,159.321
C03214=1021.708,97.418,390.551,167.495,50.393,159.322
C03215=1021.702,97.170,390.570,167.493,50.399,159.322
C03216=1021.697,96.920,390.588,167.490,50.405,159.323
C03217=1021.691,96.671,390.606,167.487,50.411,159.324
C03218=1021.686,96.422,390.623,167.484,50.417,159.324
C03219=1021.680,96.172,390.643,167.481,50.422,159.325
C03220=1021.675,95.923,390.660,167.478,50.428,159.326
C03221=1021.668,95.674,390.678,167.476,50.434,159.326
C03222=1021.664,95.424,390.696,167.474,50.439,159.327
C03223=1021.657,95.175,390.715,167.471,50.445,159.328
C03224=1021.652,94.926,390.732,167.468,50.451,159.328
C03225=1021.647,94.677,390.751,167.465,50.457,159.329
C03226=1021.641,94.427,390.769,167.462,50.462,159.329
C03227=1021.635,94.179,390.787,167.460,50.468,159.330
C03228=1021.629,93.929,390.805,167.457,50.474,159.331
C03229=1021.624,93.679,390.823,167.455,50.479,159.332
C03230=1021.618,93.430,390.841,167.452,50.485,159.332
C03231=1021.612,93.181,390.859,167.449,50.491,159.333
C03232=1021.607,92.932,390.877,167.446,50.497,159.333
C03233=1021.601,92.682,390.895,167.444,50.502,159.334
C03234=1021.596,92.433,390.913,167.441,50.507,159.335
C03235=1021.591,92.184,390.931,167.438,50.513,159.335
C03236=1021.585,91.934,390.949,167.435,50.519,159.336
C03237=1021.578,91.651,390.970,167.433,50.525,159.337
C03238=1021.572,91.368,390.990,167.429,50.532,159.338
C03239=1021.566,91.084,391.011,167.426,50.538,159.338
C03240=1021.559,90.801,391.031,167.423,50.545,159.339
C03241=1021.554,90.552,391.049,167.420,50.551,159.340
C03242=1021.548,90.303,391.067,167.418,50.556,159.340
C03243=1021.542,90.053,391.085,167.415,50.562,159.341
C03244=1021.537,89.804,391.103,167.413,50.568,159.342
C03245=1021.532,89.555,391.120,167.409,50.573,159.342
C03246=1021.526,89.305,391.138,167.406,50.579,159.343
C03247=1021.521,89.056,391.156,167.405,50.584,159.343
C03248=1021.515,88.807,391.174,167.402,50.590,159.344
C03249=1021.509,88.557,391.192,167.399,50.596,159.345
C03250=1021.503,88.308,391.209,167.396,50.601,159.345
C03251=1021.497,88.058,391.227,167.393,50.607,159.346
C03252=1021.491,87.809,391.244,167.390,50.613,159.347
C03253=1021.486,87.560,391.262,167.388,50.619,159.347
C03254=1021.480,87.311,391.280,167.385,50.625,159.348
C03255=1021.474,87.062,391.297,167.383,50.631,159.349
C03256=1021.469,86.813,391.315,167.380,50.637,159.350
C03257=1021.463,86.563,391.333,167.378,50.642,159.350
C03258=1021.457,86.314,391.350,167.375,50.648,159.351
C03259=1021.452,86.065,391.368,167.372,50.654,159.351
C03260=1021.446,85.815,391.385,167.369,50.660,159.352
C03261=1021.440,85.565,391.403,167.366,50.666,159.353
C03262=1021.435,85.316,391.420,167.365,50.671,159.354
C03263=1021.429,85.067,391.438,167.362,50.677,159.354
C03264=1021.423,84.818,391.456,167.358,50.682,159.355
C03265=1021.418,84.569,391.473,167.356,50.688,159.355
C03266=1021.412,84.319,391.491,167.353,50.694,159.356
C03267=1021.407,84.070,391.509,167.350,50.700,159.357
C03268=1021.401,83.820,391.526,167.348,50.705,159.357
C03269=1021.395,83.571,391.543,167.345,50.711,159.358
C03270=1021.390,83.322,391.561,167.343,50.717,159.359
C03271=1021.384,83.072,391.579,167.340,50.723,159.359
C03272=1021.378,82.823,391.596,167.337,50.728,159.360
C03273=1021.373,82.574,391.614,167.334,50.734,159.360
C03274=1021.367,82.325,391.631,167.332,50.740,159.361
C03275=1021.361,82.075,391.649,167.329,50.745,159.362
C03276=1021.356,81.826,391.666,167.327,50.751,159.363
C03277=1021.350,81.577,391.684,167.324,50.757,159.363
C03278=1021.345,81.328,391.701,167.321,50.763,159.364
C03279=1021.339,81.078,391.718,167.319,50.768,159.365
C03280=1021.333,80.828,391.736,167.316,50.774,159.365
C03281=1021.328,80.579,391.754,167.313,50.779,159.366
C03282=1021.322,80.330,391.771,167.310,50.785,159.366
C03283=1021.317,80.081,391.788,167.307,50.791,159.367
C03284=1021.311,79.831,391.806,167.306,50.797,159.368
C03285=1021.305,79.582,391.824,167.303,50.802,159.368
C03286=1021.300,79.333,391.841,167.300,50.808,159.369
C03287=1021.295,79.083,391.858,167.297,50.814,159.370
C03288=1021.289,78.834,391.876,167.294,50.819,159.370
C03289=1021.284,78.585,391.893,167.292,50.825,159.371
C03290=1021.278,78.335,391.911,167.289,50.830,159.371
C03291=1021.272,78.086,391.928,167.287,50.836,159.372
C03292=1021.267,77.836,391.946,167.284,50.842,159.373
C03293=1021.261,77.587,391.963,167.282,50.848,159.373
C03294=1021.255,77.338,391.979,167.279,50.853,159.374
C03295=1021.249,77.088,391.997,167.276,50.859,159.375
C03296=1021.244,76.839,392.015,167.273,50.864,159.375
C03297=1021.239,76.590,392.032,167.270,50.870,159.376
C03298=1021.233,76.341,392.049,167.268,50.876,159.376
C03299=1021.227,76.091,392.066,167.266,50.882,159.377
C03300=1021.222,75.842,392.083,167.263,50.887,159.378
C03301=1021.215,75.559,392.103,167.260,50.894,159.379
C03302=1021.209,75.275,392.122,167.257,50.901,159.379
C03303=1021.202,74.992,392.141,167.253,50.907,159.380
C03304=1021.196,74.708,392.161,167.251,50.914,159.381
C03305=1021.190,74.459,392.178,167.248,50.919,159.381
C03306=1021.184,74.210,392.195,167.245,50.925,159.382
C03307=1021.179,73.961,392.212,167.243,50.931,159.383
C03308=1021.173,73.711,392.229,167.241,50.937,159.384
C03309=1021.167,73.462,392.246,167.238,50.943,159.384
C03310=1021.161,73.212,392.263,167.235,50.948,159.385
C03311=1021.156,72.963,392.281,167.232,50.954,159.385
C03312=1021.150,72.714,392.297,167.230,50.960,159.386
C03313=1021.144,72.465,392.315,167.227,50.966,159.387
C03314=1021.139,72.215,392.331,167.225,50.971,159.387
C03315=1021.133,71.966,392.348,167.222,50.977,159.388
C03316=1021.128,71.717,392.365,167.219,50.982,159.389
C03317=1021.122,71.466,392.382,167.216,50.988,159.389
C03318=1021.116,71.217,392.400,167.213,50.994,159.390
C03319=1021.110,70.968,392.416,167.212,51.000,159.391
C03320=1021.105,70.719,392.434,167.209,51.006,159.391
C03321=1021.099,70.470,392.450,167.206,51.011,159.392
C03322=1021.094,70.220,392.467,167.203,51.017,159.393
C03323=1021.088,69.971,392.485,167.200,51.023,159.393
C03324=1021.082,69.722,392.501,167.198,51.028,159.394
C03325=1021.077,69.472,392.518,167.196,51.034,159.394
C03326=1021.071,69.223,392.535,167.193,51.040,159.395
C03327=1021.066,68.974,392.551,167.190,51.045,159.396
C03328=1021.060,68.724,392.568,167.187,51.051,159.396
C03329=1021.055,68.475,392.586,167.185,51.057,159.397
C03330=1021.049,68.225,392.602,167.183,51.063,159.398
C03331=1021.044,67.976,392.619,167.180,51.069,159.398
C03332=1021.037,67.726,392.636,167.177,51.074,159.399
C03333=1021.032,67.477,392.653,167.174,51.080,159.399
C03334=1021.026,67.227,392.669,167.172,51.085,159.400
C03335=1021.020,66.978,392.686,167.169,51.091,159.401
C03336=1021.014,66.729,392.703,167.167,51.097,159.401
C03337=1021.009,66.479,392.720,167.164,51.103,159.402
C03338=1021.003,66.230,392.736,167.161,51.109,159.403
C03339=1020.998,65.980,392.753,167.158,51.115,159.403
C03340=1020.992,65.731,392.769,167.156,51.120,159.404
C03341=1020.986,65.482,392.786,167.154,51.126,159.405
C03342=1020.980,65.233,392.803,167.151,51.132,159.405
C03343=1020.974,64.983,392.820,167.148,51.137,159.406
C03344=1020.969,64.734,392.836,167.145,51.143,159.406
C03345=1020.963,64.484,392.853,167.143,51.148,159.407
C03346=1020.958,64.235,392.870,167.140,51.154,159.408
C03347=1020.952,63.986,392.887,167.138,51.160,159.408
C03348=1020.946,63.736,392.903,167.135,51.166,159.409
C03349=1020.941,63.487,392.920,167.132,51.172,159.410
C03350=1020.935,63.237,392.936,167.130,51.177,159.411
C03351=1020.929,62.988,392.953,167.127,51.183,159.411
C03352=1020.923,62.738,392.969,167.124,51.188,159.412
C03353=1020.918,62.489,392.985,167.122,51.195,159.412
C03354=1020.912,62.240,393.001,167.119,51.201,159.413
C03355=1020.906,61.990,393.018,167.117,51.207,159.414
C03356=1020.900,61.741,393.035,167.114,51.213,159.414
C03357=1020.894,61.491,393.051,167.111,51.219,159.415
C03358=1020.889,61.242,393.067,167.108,51.224,159.416
C03359=1020.883,60.993,393.083,167.107,51.230,159.416
C03360=1020.877,60.743,393.100,167.104,51.236,159.417
C03361=1020.871,60.494,393.116,167.101,51.242,159.418
C03362=1020.865,60.245,393.132,167.098,51.248,159.418
C03363=1020.859,59.995,393.148,167.095,51.254,159.419
C03364=1020.854,59.746,393.165,167.093,51.259,159.420
C03365=1020.847,59.462,393.183,167.090,51.266,159.420
C03366=1020.840,59.178,393.202,167.087,51.272,159.421
C03367=1020.833,58.896,393.220,167.084,51.279,159.422
C03368=1020.828,58.612,393.238,167.081,51.286,159.422
C03369=1020.822,58.363,393.254,167.078,51.292,159.423
C03370=1020.816,58.114,393.271,167.075,51.298,159.424
C03371=1020.810,57.864,393.287,167.073,51.303,159.424
C03372=1020.804,57.615,393.303,167.071,51.309,159.425
C03373=1020.799,57.365,393.319,167.068,51.315,159.426
C03374=1020.793,57.115,393.336,167.065,51.321,159.426
C03375=1020.787,56.866,393.352,167.062,51.326,159.427
C03376=1020.781,56.617,393.368,167.059,51.332,159.428
C03377=1020.775,56.367,393.384,167.057,51.338,159.428
C03378=1020.770,56.119,393.400,167.055,51.343,159.429
C03379=1020.764,55.869,393.416,167.052,51.349,159.430
C03380=1020.758,55.619,393.432,167.049,51.355,159.430
C03381=1020.753,55.370,393.449,167.047,51.361,159.431
C03382=1020.747,55.120,393.465,167.044,51.367,159.431
C03383=1020.741,54.871,393.481,167.041,51.373,159.432
C03384=1020.735,54.622,393.498,167.040,51.378,159.433
C03385=1020.729,54.372,393.513,167.036,51.384,159.433
C03386=1020.724,54.123,393.529,167.034,51.390,159.434
C03387=1020.718,53.874,393.545,167.031,51.395,159.435
C03388=1020.712,53.624,393.562,167.028,51.401,159.435
C03389=1020.706,53.374,393.577,167.025,51.407,159.436
C03390=1020.701,53.125,393.594,167.024,51.413,159.437
C03391=1020.695,52.875,393.610,167.021,51.418,159.437
C03392=1020.690,52.627,393.626,167.018,51.424,159.438
C03393=1020.684,52.377,393.642,167.015,51.430,159.438
C03394=1020.678,52.127,393.658,167.012,51.436,159.439
C03395=1020.672,51.878,393.674,167.011,51.441,159.440
C03396=1020.666,51.629,393.690,167.008,51.447,159.440
C03397=1020.661,51.379,393.706,167.005,51.452,159.441
C03398=1020.655,51.130,393.722,167.002,51.458,159.441
C03399=1020.650,50.880,393.739,166.999,51.464,159.442
C03400=1020.644,50.631,393.755,166.998,51.470,159.443
C03401=1020.639,50.381,393.771,166.994,51.475,159.443
C03402=1020.633,50.132,393.786,166.992,51.481,159.444
C03403=1020.627,49.883,393.803,166.989,51.487,159.444
C03404=1020.622,49.633,393.818,166.986,51.493,159.445
C03405=1020.616,49.384,393.834,166.985,51.498,159.446
C03406=1020.610,49.134,393.851,166.981,51.504,159.446
C03407=1020.605,48.885,393.866,166.979,51.510,159.447
C03408=1020.599,48.636,393.882,166.976,51.516,159.448
C03409=1020.594,48.386,393.899,166.974,51.520,159.448
C03410=1020.588,48.136,393.915,166.971,51.526,159.449
C03411=1020.583,47.887,393.930,166.968,51.532,159.449
C03412=1020.577,47.638,393.947,166.966,51.538,159.450
C03413=1020.571,47.388,393.962,166.964,51.543,159.451
C03414=1020.565,47.139,393.978,166.961,51.549,159.451
C03415=1020.560,46.890,393.994,166.958,51.555,159.452
C03416=1020.554,46.640,394.010,166.955,51.560,159.452
C03417=1020.548,46.391,394.026,166.952,51.566,159.453
C03418=1020.543,46.142,394.041,166.951,51.572,159.454
C03419=1020.537,45.892,394.058,166.947,51.577,159.454
C03420=1020.532,45.642,394.074,166.945,51.583,159.455
C03421=1020.526,45.393,394.090,166.942,51.589,159.455
C03422=1020.521,45.143,394.105,166.940,51.594,159.456
C03423=1020.515,44.894,394.121,166.937,51.600,159.457
C03424=1020.509,44.645,394.138,166.934,51.605,159.457
C03425=1020.504,44.395,394.153,166.932,51.610,159.458
C03426=1020.498,44.146,394.169,166.930,51.616,159.458
C03427=1020.493,43.896,394.185,166.927,51.622,159.459
C03428=1020.487,43.647,394.201,166.924,51.627,159.459
C03429=1020.481,43.363,394.219,166.921,51.634,159.460
C03430=1020.474,43.080,394.237,166.919,51.640,159.461
C03431=1020.469,42.796,394.254,166.915,51.646,159.461
C03432=1020.463,42.512,394.273,166.913,51.653,159.462
C03433=1020.456,42.263,394.288,166.910,51.658,159.463
C03434=1020.450,42.013,394.304,166.907,51.664,159.463
C03435=1020.445,41.764,394.319,166.904,51.670,159.464
C03436=1020.439,41.515,394.335,166.902,51.676,159.465
C03437=1020.434,41.265,394.351,166.899,51.681,159.465
C03438=1020.428,41.016,394.365,166.897,51.687,159.466
C03439=1020.422,40.767,394.382,166.894,51.693,159.466
C03440=1020.417,40.517,394.397,166.891,51.699,159.467
C03441=1020.411,40.267,394.412,166.889,51.704,159.468
C03442=1020.405,40.018,394.429,166.886,51.710,159.468
C03443=1020.400,39.769,394.443,166.884,51.716,159.469
C03444=1020.394,39.519,394.459,166.881,51.721,159.469
C03445=1020.388,39.270,394.475,166.878,51.727,159.470
C03446=1020.383,39.020,394.490,166.876,51.732,159.471
C03447=1020.377,38.770,394.506,166.874,51.738,159.471
C03448=1020.371,38.522,394.521,166.870,51.744,159.472
C03449=1020.366,38.272,394.537,166.868,51.749,159.472
C03450=1020.360,38.022,394.552,166.865,51.755,159.473
C03451=1020.355,37.773,394.567,166.863,51.760,159.474
C03452=1020.349,37.524,394.584,166.860,51.766,159.474
C03453=1020.343,37.274,394.598,166.858,51.772,159.475
C03454=1020.337,37.025,394.614,166.854,51.778,159.475
C03455=1020.332,36.775,394.629,166.853,51.783,159.476
C03456=1020.327,36.525,394.644,166.850,51.789,159.477
C03457=1020.320,36.276,394.660,166.847,51.794,159.477
C03458=1020.314,36.026,394.676,166.844,51.800,159.478
C03459=1020.309,35.777,394.690,166.842,51.806,159.478
C03460=1020.303,35.527,394.706,166.839,51.812,159.479
C03461=1020.297,35.279,394.720,166.837,51.817,159.480
C03462=1020.292,35.029,394.736,166.834,51.823,159.480
C03463=1020.287,34.779,394.751,166.831,51.829,159.481
C03464=1020.280,34.530,394.766,166.829,51.835,159.481
C03465=1020.275,34.280,394.781,166.826,51.840,159.482
C03466=1020.269,34.031,394.796,166.823,51.846,159.482
C03467=1020.263,33.781,394.812,166.820,51.852,159.483
C03468=1020.257,33.532,394.827,166.819,51.858,159.484
C03469=1020.251,33.282,394.842,166.816,51.863,159.484
C03470=1020.246,33.033,394.857,166.813,51.869,159.485
C03471=1020.240,32.784,394.873,166.810,51.875,159.486
C03472=1020.234,32.535,394.887,166.807,51.881,159.486
C03473=1020.229,32.285,394.903,166.805,51.886,159.487
C03474=1020.223,32.035,394.918,166.803,51.892,159.487
C03475=1020.217,31.786,394.933,166.800,51.898,159.488
C03476=1020.212,31.536,394.948,166.797,51.903,159.488
C03477=1020.206,31.287,394.963,166.794,51.909,159.489
C03478=1020.201,31.037,394.978,166.792,51.915,159.490
C03479=1020.194,30.788,394.993,166.790,51.920,159.490
C03480=1020.189,30.539,395.008,166.787,51.926,159.491
C03481=1020.183,30.289,395.023,166.784,51.932,159.492
C03482=1020.178,30.040,395.038,166.781,51.937,159.492
C03483=1020.171,29.790,395.053,166.778,51.943,159.493
C03484=1020.166,29.541,395.068,166.776,51.948,159.493
C03485=1020.160,29.291,395.083,166.774,51.954,159.494
C03486=1020.155,29.042,395.099,166.771,51.960,159.494
C03487=1020.149,28.792,395.114,166.768,51.965,159.495
C03488=1020.143,28.543,395.129,166.765,51.971,159.495
C03489=1020.138,28.292,395.144,166.764,51.977,159.496
C03490=1020.132,28.043,395.158,166.761,51.982,159.497
C03491=1020.127,27.793,395.174,166.758,51.988,159.497
C03492=1020.121,27.544,395.188,166.755,51.993,159.498
C03493=1020.115,27.261,395.205,166.752,52.000,159.499
C03494=1020.108,26.977,395.222,166.749,52.007,159.499
C03495=1020.101,26.693,395.238,166.747,52.013,159.500
C03496=1020.095,26.410,395.255,166.743,52.020,159.500
C03497=1020.089,26.160,395.271,166.740,52.026,159.501
C03498=1020.083,25.911,395.286,166.738,52.030,159.502
C03499=1020.078,25.662,395.300,166.735,52.036,159.502
C03500=1020.072,25.412,395.316,166.733,52.042,159.503
C03501=1020.067,25.162,395.330,166.730,52.048,159.503
C03502=1020.060,24.912,395.344,166.727,52.054,159.504
C03503=1020.054,24.664,395.359,166.724,52.060,159.504
C03504=1020.049,24.413,395.374,166.721,52.065,159.505
C03505=1020.043,24.164,395.388,166.720,52.071,159.506
C03506=1020.037,23.915,395.403,166.717,52.077,159.506
C03507=1020.032,23.665,395.419,166.714,52.082,159.507
C03508=1020.026,23.415,395.432,166.711,52.088,159.507
C03509=1020.021,23.167,395.447,166.709,52.094,159.508
C03510=1020.014,22.917,395.462,166.706,52.099,159.508
C03511=1020.009,22.667,395.476,166.704,52.105,159.509
C03512=1020.003,22.417,395.491,166.701,52.111,159.510
C03513=1019.997,22.168,395.506,166.698,52.116,159.510
C03514=1019.993,21.918,395.520,166.696,52.122,159.511
C03515=1019.986,21.669,395.535,166.692,52.127,159.511
C03516=1019.980,21.420,395.550,166.690,52.133,159.512
C03517=1019.975,21.170,395.564,166.688,52.139,159.513
C03518=1019.969,20.920,395.579,166.685,52.144,159.513
C03519=1019.963,20.671,395.594,166.682,52.150,159.514
C03520=1019.958,20.422,395.608,166.679,52.156,159.514
C03521=1019.952,20.172,395.623,166.677,52.162,159.515
C03522=1019.947,19.923,395.638,166.675,52.167,159.515
C03523=1019.941,19.673,395.652,166.672,52.173,159.516
C03524=1019.935,19.424,395.667,166.669,52.178,159.516
C03525=1019.930,19.174,395.681,166.666,52.184,159.517
C03526=1019.924,18.925,395.696,166.664,52.190,159.518
C03527=1019.918,18.675,395.710,166.661,52.195,159.518
C03528=1019.912,18.426,395.725,166.659,52.201,159.519
C03529=1019.907,18.176,395.738,166.656,52.206,159.519
C03530=1019.900,17.926,395.753,166.653,52.212,159.520
C03531=1019.895,17.677,395.767,166.651,52.218,159.520
C03532=1019.890,17.427,395.782,166.648,52.224,159.521
C03533=1019.884,17.177,395.797,166.645,52.230,159.521
C03534=1019.878,16.928,395.811,166.643,52.234,159.522
C03535=1019.873,16.679,395.825,166.640,52.241,159.523
C03536=1019.867,16.430,395.840,166.637,52.246,159.523
C03537=1019.861,16.179,395.854,166.635,52.252,159.524
C03538=1019.855,15.930,395.868,166.632,52.258,159.524
C03539=1019.849,15.681,395.882,166.629,52.263,159.525
C03540=1019.844,15.432,395.898,166.627,52.269,159.526
C03541=1019.838,15.181,395.912,166.624,52.274,159.526
C03542=1019.833,14.932,395.926,166.622,52.280,159.527
C03543=1019.827,14.683,395.940,166.618,52.285,159.527
C03544=1019.822,14.433,395.954,166.616,52.291,159.528
C03545=1019.815,14.184,395.969,166.613,52.297,159.528
C03546=1019.810,13.934,395.983,166.611,52.302,159.529
C03547=1019.804,13.684,395.997,166.608,52.308,159.529
C03548=1019.798,13.436,396.011,166.606,52.314,159.530
C03549=1019.792,13.185,396.026,166.602,52.319,159.530
C03550=1019.787,12.936,396.039,166.600,52.325,159.531
C03551=1019.781,12.687,396.054,166.597,52.331,159.531
C03552=1019.776,12.437,396.068,166.594,52.336,159.532
C03553=1019.770,12.187,396.082,166.592,52.343,159.533
C03554=1019.764,11.937,396.096,166.588,52.348,159.533
C03555=1019.758,11.689,396.110,166.587,52.354,159.534
C03556=1019.752,11.439,396.124,166.584,52.360,159.534
C03557=1019.746,11.156,396.140,166.581,52.366,159.535
C03558=1019.740,10.874,396.155,166.578,52.372,159.535
C03559=1019.732,10.592,396.171,166.575,52.379,159.536
C03560=1019.726,10.310,396.187,166.571,52.385,159.537
C03561=1019.720,10.060,396.201,166.569,52.391,159.537
C03562=1019.715,9.811,396.215,166.566,52.396,159.538
C03563=1019.709,9.561,396.228,166.564,52.402,159.538
C03564=1019.703,9.312,396.243,166.561,52.408,159.539
C03565=1019.697,9.063,396.257,166.558,52.414,159.540
C03566=1019.692,8.813,396.271,166.556,52.420,159.540
C03567=1019.686,8.563,396.285,166.552,52.425,159.541
C03568=1019.680,8.313,396.299,166.550,52.431,159.541
C03569=1019.674,8.064,396.312,166.547,52.437,159.542
C03570=1019.669,7.814,396.326,166.545,52.442,159.542
C03571=1019.663,7.566,396.341,166.542,52.448,159.543
C03572=1019.657,7.316,396.354,166.540,52.454,159.543
C03573=1019.652,7.066,396.368,166.537,52.459,159.544
C03574=1019.645,6.816,396.382,166.534,52.465,159.544
C03575=1019.640,6.567,396.396,166.531,52.470,159.545
C03576=1019.634,6.317,396.410,166.528,52.476,159.545
C03577=1019.629,6.068,396.424,166.526,52.481,159.546
C03578=1019.623,5.818,396.437,166.524,52.487,159.547
C03579=1019.618,5.569,396.451,166.521,52.493,159.547
C03580=1019.611,5.319,396.465,166.518,52.499,159.548
C03581=1019.606,5.070,396.478,166.515,52.504,159.548
C03582=1019.601,4.820,396.492,166.512,52.510,159.549
C03583=1019.594,4.570,396.507,166.509,52.516,159.549
C03584=1019.589,4.320,396.520,166.508,52.521,159.550
C03585=1019.583,4.071,396.534,166.505,52.527,159.550
C03586=1019.577,3.821,396.547,166.502,52.532,159.551
C03587=1019.572,3.572,396.561,166.499,52.538,159.551
C03588=1019.566,3.322,396.575,166.496,52.543,159.552
C03589=1019.561,3.073,396.589,166.493,52.549,159.552
C03590=1019.555,2.823,396.602,166.490,52.555,159.553
C03591=1019.549,2.574,396.616,166.488,52.560,159.553
C03592=1019.544,2.324,396.630,166.486,52.566,159.554
C03593=1019.538,2.075,396.644,166.483,52.571,159.554
C03594=1019.533,1.825,396.658,166.480,52.577,159.555
C03595=1019.527,1.576,396.672,166.477,52.582,159.555
C03596=1019.521,1.326,396.685,166.474,52.588,159.556
C03597=1019.516,1.077,396.699,166.473,52.594,159.557
C03598=1019.510,0.827,396.713,166.469,52.599,159.557
C03599=1019.505,0.578,396.727,166.466,52.604,159.557
C03600=1019.499,0.328,396.740,166.464,52.610,159.558
C03601=1019.493,0.079,396.754,166.461,52.616,159.558
C03602=1019.487,-0.171,396.768,166.459,52.621,159.559
C03603=1019.482,-0.420,396.781,166.456,52.627,159.560
C03604=1019.477,-0.670,396.795,166.453,52.632,159.560
C03605=1019.471,-0.920,396.809,166.450,52.637,159.560
C03606=1019.465,-1.169,396.822,166.447,52.643,159.561
C03607=1019.460,-1.419,396.836,166.445,52.649,159.561
C03608=1019.454,-1.669,396.849,166.443,52.654,159.562
C03609=1019.449,-1.918,396.863,166.440,52.659,159.562
C03610=1019.442,-2.167,396.877,166.437,52.665,159.563
C03611=1019.437,-2.417,396.890,166.434,52.671,159.563
C03612=1019.432,-2.667,396.904,166.431,52.676,159.564
C03613=1019.426,-2.917,396.917,166.429,52.681,159.564
C03614=1019.421,-3.166,396.931,166.426,52.687,159.565
C03615=1019.415,-3.416,396.945,166.423,52.692,159.565
C03616=1019.409,-3.665,396.958,166.420,52.698,159.566
C03617=1019.404,-3.915,396.972,166.418,52.703,159.566
C03618=1019.399,-4.165,396.985,166.415,52.708,159.567
C03619=1019.392,-4.414,396.999,166.413,52.714,159.567
C03620=1019.387,-4.664,397.013,166.410,52.720,159.568
C03621=1019.381,-4.944,397.026,166.406,52.726,159.568
C03622=1019.374,-5.224,397.042,166.404,52.733,159.569
C03623=1019.368,-5.505,397.057,166.400,52.739,159.570
C03624=1019.361,-5.785,397.072,166.398,52.745,159.570
C03625=1019.356,-6.035,397.085,166.395,52.751,159.571
C03626=1019.350,-6.283,397.098,166.392,52.757,159.571
C03627=1019.344,-6.533,397.111,166.389,52.762,159.572
C03628=1019.339,-6.783,397.124,166.386,52.767,159.572
C03629=1019.333,-7.032,397.138,166.384,52.774,159.573
C03630=1019.327,-7.282,397.151,166.380,52.779,159.573
C03631=1019.321,-7.532,397.164,166.378,52.785,159.574
C03632=1019.316,-7.782,397.177,166.376,52.790,159.574
C03633=1019.310,-8.031,397.190,166.373,52.795,159.575
C03634=1019.304,-8.281,397.203,166.370,52.801,159.575
C03635=1019.299,-8.530,397.216,166.367,52.807,159.576
C03636=1019.293,-8.779,397.230,166.365,52.813,159.576
C03637=1019.288,-9.029,397.243,166.362,52.818,159.577
C03638=1019.281,-9.279,397.256,166.359,52.824,159.577
C03639=1019.276,-9.528,397.269,166.356,52.830,159.578
C03640=1019.270,-9.778,397.283,166.353,52.835,159.578
C03641=1019.265,-10.027,397.295,166.350,52.840,159.579
C03642=1019.259,-10.277,397.309,166.348,52.847,159.579
C03643=1019.253,-10.527,397.321,166.346,52.852,159.580
